(* IEC 61131-3 sources: ml2plc/benchmarks/st (part 23) *)

    bias_3 : ARRAY[0..63] OF REAL := [-0.00983189233, 0.0739286318, -0.03035645, 0.0550533831, -0.011248054, 0, -0.0295825377, -0.0090773385, 0, -0.0277472436, -0.00766381249, -0.00870534033, -0.0367787257, -0.0242641736, -0.00147182879, -0.00894620363, 0.0173237566, 0.00239057303, -0.00620334735, -0.00517789647, -0.0133990953, 0.0294917747, 0.0401097015, -0.0258607231, -0.00522571057, 0, -0.0150696058, 0.0860590115, -0.0117668696, 0.065539062, -0.00745888008, -0.0186666064, -0.010953215, -0.0240848884, -0.0448102988, -0.0404310934, 0.0785407722, 0.0790930837, -0.0278634299, -0.0265457965, 0, -0.0240220856, 0.00635804934, 0.0217319299, -0.02775204, 0.00820828322, 0.0399322994, 0.0746404901, -0.0329935588, 0, 0.00812079571, -0.0131024169, -0.0233938117, 0.0117759928, 0.0732261613, -0.0248215012, 0, 0.000535005063, 0.0062644016, 0.0363470353, 0.0787089318, -0.0285863206, 0, 0.0387545452];

    weights_6 : ARRAY[0..4095] OF REAL := [-0.0211104695, 0.157233626, 0.0721651465, -0.0791621804, -0.145463645, 0.0476885587, 0.103807047, -0.217098057, 0.15736191, -0.173330665, -0.128692865, -0.0421262085, 0.0980989784, 0.155999586, 0.0207046866, 0.184844807, -0.00715442142, 0.172988996, -0.206348658, 0.157887205, -0.037524119, -0.140499547, 0.187242225, 0.152909175, -0.145436138, -0.0675008371, 0.169665024, 0.210023656, 0.206236467, 0.208556831, 0.0959817022, -0.148986042, 0.0728623122, 0.026120171, 0.211910024, -0.0622561015, 0.0902522206, 0.0471122339, 0.0779013783, 0.0172086973, -0.039685376, -0.0467820168, 0.0570690036, 0.0242511332, -0.209991112, 0.00939850137, 0.112361535, 0.116925567, -0.153550565, 0.212469026, 0.14040117, -0.0208477583, 0.182546362, 0.0197014436, 0.186374202, -0.168809876, 0.196177915, -0.00232131779, 0.137093261, 0.162052512, 0.199661002, 0.0766961128, 0.211054429, 0.125300422, 0.00426613819, 0.288283914, -0.159290671, -0.0769464672, 0.0940423161, -0.0546351485, 0.0653043687, 0.0303289033, 0.0641354099, -0.192860484, 0.04200764, 0.0343205296, 0.155289501, -0.180832982, -0.12778616, 0.262020022, 0.0602597371, 0.10863255, -0.237889618, -0.095524922, -0.272757202, -0.0731869787, -0.0907882899, -0.147379801, -0.169592246, 0.178864881, -0.101507559, -0.0397703201, 0.016668126, 0.0635820627, 0.0767925531, -0.102012202, 0.0477126874, 0.0524956584, 0.111083403, -0.0878348276, 0.011967063, -0.0565153994, 0.170608982, 0.309960365, -0.105272628, 0.211850211, -0.0994742885, -0.153632715, 0.267046332, -0.203152657, -0.160044357, 0.0353948474, -0.0975862592, -0.0403899029, 0.07099244, 0.0249471422, -0.0422067828, -0.220276818, -0.185284197, -0.0370966718, 0.148172244, -0.120848358, -0.0141801946, -0.0953512639, -0.253198028, 0.104871087, 0.0740961581, -0.182465032, 0.0539166033, -0.159959942, -0.161966518, 0.0288212746, -0.135103494, -0.112145692, -0.0749802366, -0.0615305528, 0.157502532, 0.0857658535, -0.0273212269, 0.141590878, -0.0330497138, 0.176339731, -0.0418806784, 0.0999175385, -0.0713153332, 0.263013691, -0.115717605, 0.204661101, -0.11504811, -0.0947428197, 0.153199002, 0.335939616, -0.00631709397, 0.100122802, -0.209013268, 0.0137379616, -0.204656497, 0.0605559498, -0.175298169, -0.123451911, -0.0473049544, 0.0416926257, 0.156591177, -0.101554133, 0.115582488, -0.0190878287, -0.0975746512, 0.155756831, 0.108877532, 0.171931863, 0.235213891, 0.00560221262, -0.151249588, 0.00370491436, -0.0536345989, -0.181572989, -0.117012545, -0.106260225, 0.242837548, 0.223648071, 0.0628157556, 0.295081288, -0.0346996188, 0.15143846, 0.187727511, 0.290291816, 0.0033030943, -0.161266476, 0.00898908544, 0.244648784, -0.134097993, 0.0367004983, 0.0216495004, 0.180981815, -0.0798874199, 0.13122049, 0.0334438831, 0.0200074967, 0.103910699, -0.102675296, -0.207296401, 0.0869636759, -0.20655781, -0.0956464559, -0.203777537, -0.105265148, 0.0783180222, -0.0458374731, 0.204411358, 0.118474796, 0.122315288, -0.0419053994, -0.340604126, 0.135242134, -0.129586041, -0.0497838371, -0.0099619776, -0.0477824807, 0.281962305, 0.00426848233, -0.181631833, -0.170377254, 0.104996637, 0.114299156, -0.163810551, 0.249239355, -0.0833768472, 0.0697716847, 0.014485863, 0.157567188, 0.110193223, 0.230861947, -0.110680073, -0.0243154187, -0.0779362693, -0.0843363702, -0.049658794, -0.00124949845, -0.0668900907, 0.086151801, 0.179528475, 0.0938131064, -0.204934552, 0.0532739088, -0.120318048, -0.151893049, -0.146782264, 0.312886775, 0.0673337728, -0.1004811, -0.171645507, 0.268849701, -0.229744852, -0.134535402, -0.119718812, 0.0152729712, -0.196205392, -0.123321056, 0.00104016194, 0.114403293, -0.109209985, -0.116009399, -0.00587476185, -0.100333177, 0.104191698, 0.0102303922, -0.134384453, -0.204718813, 0.0862976313, 0.140776381, 0.0467067696, 0.094970122, -0.189605281, -0.0276639797, -0.0749640316, 0.0723377988, 0.00538966572, 0.0190833975, -0.0198820475, -0.00954220816, 0.0676214248, 0.104344197, -0.200903356, -0.206617773, 0.084322378, -0.0795044377, -0.0956577435, 0.191447124, -0.0795495212, -0.00805467833, 0.205130324, 0.179273605, -0.0990068316, -0.0614028908, 0.148120746, 0.132912666, -0.189888284, 0.200087667, -0.164052576, -0.0751432627, 0.0476862341, 0.0292347074, -0.052457124, -0.0892619789, 0.0716815516, 0.0529787801, 0.213911965, 0.209351331, -0.129100218, 0.0809682086, 0.176059052, 0.149538949, -0.126543701, -0.188590631, -0.183877945, 0.117343932, -0.167362183, -0.0124702444, -0.152586102, -0.18852441, 0.0780072361, -0.153538495, 0.0840239376, -0.148158073, 0.0951781124, -0.0676086247, -0.202492416, -0.0601291209, 0.0147494972, -0.148133397, -0.00998263061, -0.096799612, -0.00623972714, -0.0822741985, 0.134943768, 0.196010545, 0.0348980874, 0.194250599, 0.00896206498, -0.170046642, 0.0372118801, 0.0163984746, 0.179545149, 0.112079129, -0.104169428, -0.0681873262, -0.14190802, -0.167659834, 0.171136335, 0.176123098, 0.15911971, -0.0608612299, -0.0210849196, -0.132437974, 0.0952331275, -0.0566280484, -0.179609761, -0.202228233, 0.160658821, -0.127846152, -0.169803977, 0.0259776413, -0.175173402, 0.108989462, -0.174509123, 0.163906083, -0.0123733133, -0.192176595, 0.168579057, 0.167967841, -0.0916754827, -0.00778664649, -0.041722253, -0.215875, 0.107255802, 0.09431611, 0.110112235, 0.155124173, -0.0552193671, -0.00624886155, -0.116997302, 0.125487968, 0.149071887, 0.0814684778, -0.0264531672, -0.202291474, -0.107270196, 0.208046228, 0.198929116, 0.124986812, -0.116254002, 0.106430285, 0.0689994991, 0.123037621, -0.144080907, 0.0291826203, -0.0867067724, -0.122828558, -0.193552107, 0.180794746, -0.151306659, -0.108268835, 0.0360157453, -0.162983239, 0.180829659, 0.123341292, -0.143707618, -0.0218093451, 0.100755021, 0.048000399, 0.0416897722, -0.030838713, -0.10653317, 0.0873832777, -0.188493058, -0.0422797352, 0.0743354112, -0.125618383, 0.163786501, -0.184897706, 0.0689249486, 0.216842949, -0.173285306, 0.185100108, -0.117793359, -0.19082053, -0.106456965, -0.0742470324, -0.0494265445, 0.165998891, -0.185700104, -0.121370681, -0.174497947, -0.0514864251, 0.10049998, -0.107571743, 0.159631327, 0.187085122, 0.0653448254, -0.120375261, 0.275558501, 0.182469591, -0.175698802, -0.0759939849, 0.065009132, 0.259765774, -0.086910978, 0.0502287, -0.0737552643, -0.0215020366, 0.161072969, 0.123396195, -0.175406262, 0.0518808141, -0.0351930261, 0.0470791981, 0.262363374, 0.1363094, 0.180866018, 0.132682219, 0.165143073, 0.126118854, 0.0938046128, -0.254130632, 0.0568571538, -0.0724096671, 0.0160691887, -0.0521572456, 0.22484374, -0.0792442709, -0.00761091337, 0.276181072, -0.086371094, -0.129833862, -0.0362726077, -0.0417017639, 0.0206526667, 0.239292666, -0.0601968914, 0.0359402746, 0.308184862, 0.0270620137, -0.208643079, 0.131217003, 0.0645703152, 0.118619733, 0.0201364737, -0.165239125, 0.162001967, 0.177479923, -0.111770749, 0.135645315, 0.0129162921, -0.202752113, -0.0295399278, 0.022838518, -0.0796107128, 0.0467211269, -0.051113341, 0.160861671, 0.00665348954, -0.104955673, -0.0838543624, -0.236661151, 0.214804575, -0.0623946115, 0.140443742, -0.0886547342, 0.0746734887, 0.276039749, -0.199886113, 0.121124074, 0.0216602683, -0.167079479, -0.138646215, -0.0189068019, -0.0126770437, 0.0390007943, 0.0360741764, -0.141568631, -0.0118533075, 0.178898349, -0.0807059556, 0.0550475866, 0.178213313, -0.0915158764, -0.109646633, -0.066618517, -0.00931756198, -0.201538652, 0.0959077924, -0.019727543, 0.00191234052, 0.180038348, 0.112552777, 0.101054952, 0.215217724, -0.185405463, 0.122277573, -0.0108845085, -0.0374378562, -0.0693836063, 0.206913039, -0.193783402, -0.0592647493, -0.198673338, -0.00192482769, -0.00480589271, 0.0151784569, -0.11449635, 0.150387093, -0.0220891237, -0.0531173348, 0.0558237582, -0.0155561566, 0.110152856, -0.10219758, 0.125887617, 0.187418178, -0.00413711369, 0.199766979, -0.0751423836, -0.196204484, -0.163247168, 0.0657932907, 0.179478303, -0.0909180194, -0.0187031627, -0.0687615424, -0.125233293, -0.00715054572, 0.191343263, -0.140845746, -0.101612061, 0.028948009, 0.00607836246, 0.0241835825, -0.0792405158, 0.170693278, 0.121472552, -0.159257323, 0.15754503, -0.139394745, -0.044453688, -0.0742065012, 0.176449284, 0.226904213, -0.0162550025, 0.281962007, 0.141561612, -0.179304242, -0.22687985, 0.0888308734, 0.1368251, -0.215948135, 0.232278898, 0.14440532, -0.210397243, 0.0025057646, 0.257558495, 0.069859311, -0.0588960908, -0.178999975, -0.00917844474, 0.0827753693, -0.0334500261, 0.0289534777, -0.147056982, 0.18982479, -0.0401569977, -0.00673311763, 0.117641859, 0.0199112538, -0.110949092, -0.10525246, -0.110742055, -0.149034083, 0.176191643, 0.164675817, -0.152210981, 0.111859016, -0.0424617529, 0.070398286, 0.0940225571, 0.160483241, -0.166004077, -0.0361319557, 0.156162739, 0.255399585, -0.0411905348, 0.0899951607, -0.214364231, -0.0514262058, 0.136874646, -0.0144281425, 0.0158658996, 0.173274562, -0.0837578475, -0.021164313, 0.189715445, 0.0227939058, 0.0768007636, 0.0420344919, 0.13114506, 0.0212835968, 0.125271335, -0.0908199325, -0.2127489, 0.223346874, -0.168397516, -0.143092021, 0.0855721906, 0.217426375, -0.010913834, 0.161978483, -0.0237388425, -0.0148029672, -0.0206773132, 0.163911536, -0.115519904, -0.0708635896, 0.160120934, 0.21680361, -0.0919932425, -0.106572457, 0.186694637, -0.0864723846, -0.0672358871, -0.0620637983, -0.0492999963, -0.031213671, -0.214064613, -0.0040052929, -0.177249506, 0.198898122, 0.029973764, 0.0648880824, -0.0722419471, 0.0583239459, -0.161417127, 0.118529066, 0.0775398463, 0.0136581725, -0.019831283, 0.0340036228, -0.069475472, -0.141518444, -0.0155703966, 0.0465259701, -0.13712129, 0.215217024, 0.153940856, 0.233599231, 0.069659397, 0.0283375084, 0.136588395, 0.114837028, 0.00435284665, -0.0815577209, 0.0850224197, 0.0896461308, 0.0839098245, 0.12630628, 0.102898523, -0.0242574364, 0.0395214707, 0.179158911, 0.140869483, -0.0315961689, -0.211324051, -0.101073779, 0.164895773, 0.0432892777, -0.0961784273, 0.187965691, -0.0886578932, -0.143109977, -0.200058162, 0.128884479, -0.150142565, -0.0212808698, -0.0118450765, 0.0831215233, -0.0732853338, -0.0489297211, 0.000687902851, 0.0266030431, -0.201587737, -0.185360029, -0.00679598097, 0.108024552, 0.102891639, -0.178852096, -0.173995063, 0.0813450366, -0.0506051332, -0.0515105948, 0.0880956501, 0.173789188, 0.00271931873, -0.181898132, -0.0750331804, -0.0916771367, 0.0279746372, -0.0858160108, 0.0492289215, -0.0897664428, 0.118924871, -0.00673155487, 0.0254511833, -0.0507416576, -0.131477594, 0.0658444315, -0.176156193, 0.00369836204, 0.209861919, -0.144315973, 0.0758810192, -0.126617879, 0.0478404015, 0.0629696399, -0.181336939, -0.070628196, 0.0589700602, 0.0671523064, 0.0530530922, 0.148497984, 0.199353352, -0.2551274, -0.155184016, -0.00421486888, 0.212831467, -0.0586378425, 0.147449061, -0.201066777, -0.0765811056, 0.0298376996, -0.028335914, -0.0145538365, 0.120011285, 0.263296843, -0.0805929601, 0.196454912, -0.194894016, 0.0144730853, 0.00976360589, 0.105623856, -0.128629684, 0.224141806, -0.244979411, 0.214529052, -0.0382702313, 0.156628206, 0.0189788435, 0.127576098, -0.204321966, -0.106341101, 0.309783638, -0.0312428474, -0.136540458, 0.271282047, -0.320485145, -0.130114317, 0.0987244472, -0.0768140033, 0.292481333, 0.028581921, 0.0651605949, 0.0565245636, -0.207960293, -0.105757877, -0.0665429085, -0.00274416106, 0.0682443231, -0.106524602, -0.163970143, 0.0532483347, -0.200977892, 0.0309002809, -0.0602365695, 0.202884033, -0.04036038, -0.0263917297, -0.138741806, 0.261350095, 0.0551347472, 0.181741431, -0.147500739, 0.178088039, 0.114219822, 0.046044156, 0.0941443816, 0.0813267976, 0.0595558062, -0.197245672, -0.0100678066, -0.211604849, -0.148000121, -0.198542699, 0.196343526, 0.138460979, 0.107107386, 0.0907673761, -0.121037595, 0.252360672, -0.0970465541, 0.0558764599, -0.0847656652, -0.209763199, 0.167329192, -0.237716049, -0.0499278046, 0.249167144, 0.0408127345, -0.165352255, 0.176838875, 0.00782003999, 0.176427022, -0.0851962119, -0.192636058, 0.187963501, 0.170646742, 0.0470952839, 0.00458228588, 0.141556203, 0.0644658133, 0.0417393818, 0.0441780165, 0.039651297, 0.0833919719, -0.172924563, 0.0634429529, -0.0965564921, 0.0724875107, 0.21937269, -0.0974312797, -0.130002752, -0.121189877, 0.0671949536, 0.0867445171, -0.00312029221, 0.126738116, 0.0653212741, 0.252740234, 0.287628323, 0.167519346, 0.139367387, -0.0309090856, 0.263746917, 0.0875785947, 0.0128881168, -0.0565036125, 0.120908678, 0.240472659, -0.201509178, 0.293792278, -0.131671205, 0.0896654353, 0.0370695144, 0.135521129, 0.20480074, -0.175205469, -0.171041086, -0.0579688512, -0.156582564, -0.0778886229, 0.0664458051, 0.130356193, 0.0996769667, -0.153313071, -0.192398816, -0.106274486, -0.0162558295, 0.0870158821, -0.192340657, 0.048169598, -0.171457037, -0.136983603, -0.064907901, 0.145346314, 0.190712199, 0.0360278338, 0.0434320495, -0.211738184, 0.160129383, -0.105414405, -0.171388596, -0.0388856754, 0.142384306, 0.137329713, -0.130360201, -0.0619715676, 0.00965698808, -0.0439127162, 0.170497492, 0.212079838, -0.142104536, 0.0586519986, -0.115233481, -0.0224351734, -0.16999881, 0.0918107182, -0.167155147, 0.195335492, -0.0757286102, -0.172540411, 0.103915311, -0.141615734, -0.00377908791, -0.0657154992, -0.148804039, 0.022908235, -0.168834493, 0.152186722, 0.0506493412, -0.112933271, 0.00049599976, 0.100557655, 0.112081513, 0.142245606, 0.0271094441, 0.0381551534, 0.20742555, -0.110420324, -0.100627325, 0.145201087, -0.202350944, 0.120480955, 0.0444104783, 0.211891606, 0.19280535, 0.0655445755, 0.189393878, 0.196804807, -0.0521670766, 0.0503715128, 0.214662924, -0.0492795333, -0.0675857663, 0.178876325, 0.0826835707, -0.169171751, 0.0269653201, 0.211806223, 0.130338058, -0.000949479057, 0.196632594, 0.186210766, 0.0524837524, -0.0555000752, -0.131404147, 0.146059439, -0.0972863659, -0.0147773847, 0.105667993, -0.00656548562, -0.144193918, 0.0886233747, 0.215485469, -0.0223604683, 0.165627271, 0.117518991, 0.000273500162, -0.196279138, 0.0528765172, 0.137227044, 0.0115529299, -0.0449971259, -0.0784725025, -0.172097519, -0.0769113824, -0.144809157, 0.087641567, 0.0567293391, -0.165308416, 0.0845244378, -0.0673978627, 0.191283584, -0.0394614935, 0.203768536, -0.202162296, -0.138682559, -0.109796427, 0.112647042, 0.0804700181, -0.0721322224, -0.102790877, -0.0195402578, 0.00424019992, -0.117378324, 0.205446005, 0.203034252, 0.101452544, -0.0454550199, 0.157199964, 0.0115054222, -0.0943236724, -0.0565667748, -0.107933104, -0.0655731708, 0.157481402, 0.128197148, 0.00223283307, -0.00375899929, -0.1018316, -0.173439905, -0.15236567, 0.212863877, -0.152796358, 0.162461266, -0.0564482771, -0.120488144, -0.13375029, 0.025584979, -0.205807254, -0.192222401, 0.214670464, -0.0954632461, 0.183467418, 0.183182776, -0.00882993639, 0.169890597, -0.197005555, -0.106948674, -0.00395756867, 0.0120129455, 0.0223759171, 0.149836347, 0.228335664, -0.0534032434, 0.132094547, -0.0133346152, 0.183536708, -0.190487862, -0.00259809522, 0.000128543412, 0.127965212, -0.0134203611, -0.129633933, 0.229406625, 0.0699569285, 0.198570237, -0.0478203781, 0.181146488, 0.0680752471, 0.00578152016, -0.110974222, -0.088077426, 0.117438272, -0.202719942, -0.0765619129, 0.0070055034, 0.00518807769, 0.0908474326, -0.210115537, -0.259739071, 0.0877127647, 0.178909853, 0.0252563711, 0.161810607, 0.14697203, 0.0207887739, 0.192217827, 0.0119345486, 0.111504808, -0.138566241, 0.0183499251, 0.178135261, 0.10215006, 0.11800538, 0.0883670896, 0.0227976646, -0.122666731, 0.0188208688, 0.0996467769, -0.100148812, 0.117532745, 0.237992808, -0.130577683, -0.15731205, 0.271030456, -0.23369348, -0.0929943994, 0.0971348509, -0.104811274, -0.120445482, -0.0412788987, 0.0163263902, 0.138564199, -0.144116297, 0.125310749, -0.172860175, -0.224062487, 0.13113521, -0.0350915194, 0.102414116, 0.00754255336, -0.0123361535, -0.0915403515, 0.0783033222, 0.109218769, 0.00511339353, 0.059927389, 0.0361303464, -0.121367157, -0.0622647256, 0.0529602021, -0.149987593, 0.0344639942, 0.244372755, -0.129179358, -0.0458081402, -0.141225874, -0.00293263793, 0.152275071, -0.0406294242, 0.139919147, 0.187548757, -0.178822875, -0.0349252298, -0.0637998432, -0.192398965, 0.0176388826, 0.0132232755, 0.081162639, 0.00220011175, -0.148068249, 0.189775273, -0.21044074, -0.193314359, -0.0609930158, -0.191583186, 0.169178709, 0.170702919, 0.149429336, 0.0734934062, -0.0319855362, 0.0536946096, 0.0498708934, -0.117750682, 0.0036894232, 0.0974819437, 0.162416473, 0.036212638, -0.152097091, 0.0102473954, -0.175146922, -0.109410793, 0.0510285608, -0.102032453, -0.0270780027, 0.112112477, 0.179075554, -0.174917683, -0.115047842, -0.104785867, 0.0759669393, -0.185626954, -0.114752382, 0.0533825904, -0.104991615, -0.0954450741, -0.0869510844, -0.132044673, -0.191752613, 0.00513811922, 0.0554652661, -0.133202344, 0.148236826, -0.174548671, 0.101005033, -0.147775263, 0.151600003, 0.195948124, 0.146968648, -0.181632847, -0.126265585, 0.0861280486, 0.0299651623, 0.0794558972, 0.0533921868, 0.0195937455, 0.0455982238, 0.150372431, 0.139378235, -0.101709567, -0.0294380337, 0.0811925083, -0.0342354178, 0.0327691734, 0.0400085896, -0.1412265, 0.0617004111, 0.0421027988, -0.104852192, 0.00592757761, -0.180350497, 0.0525539964, -0.111471675, -0.0811403841, -0.0120081007, 0.15921399, -0.188091248, 0.184693262, -0.0228968561, 0.115342319, -0.0535733849, -0.114198565, 0.0240756273, 0.147423342, 0.15892826, 0.00908050407, -0.213146105, 0.152774766, -0.00141887786, -0.0586975515, -0.114548035, 0.0891831964, -0.0406573191, 0.0181619823, -0.049714718, -0.200603843, -0.135449693, 0.129440948, -0.212808505, -0.0500480942, -0.0812454671, -0.180212289, 0.0619920045, 0.0307168979, -0.0518378466, 0.0701079816, -0.190243214, -0.138796121, -0.193981051, -0.0390182026, -0.117929213, -0.204903558, -0.202367961, -0.155948266, -0.171265543, -0.129201606, -0.0976203829, 0.221453071, 0.138735101, -0.158441961, -0.225554422, -0.0675398037, -0.132319763, -0.0978091806, 0.210110873, 0.178208128, 0.101490974, 0.0418321043, 0.160106704, -0.187610939, -0.192003295, 0.0196090881, 0.0968832597, -0.175496653, -0.0902556181, -0.155951157, 0.107045144, 0.0573832281, -0.0581211299, 0.0521087125, 0.171671689, 0.158271715, -0.212730348, -0.0388053134, -0.172507182, -0.125131086, 0.156479985, -0.335062623, -0.0702413097, 0.223254368, 0.0645823479, 0.219279632, -0.196573928, 0.0732722208, 0.263311893, -0.159265086, 0.0834448114, 0.13835384, -0.136304572, 0.106453225, -0.0613590926, 0.138230368, 0.174712658, 0.094565548, 0.0211733319, 0.102425985, 0.0467876047, 0.111685343, 0.147267804, -0.258844495, 0.145146266, 0.14244695, -0.22259891, 0.0884163454, -0.207033977, 0.202475429, 0.0740721077, -0.0818101689, -0.125599563, 0.048894804, 0.139541343, 0.0525139496, -0.179559693, -0.0716978014, 0.0090209581, 0.113008924, 0.172887772, -0.0844542906, -0.0717213899, 0.188895106, 0.00843533594, -0.161318779, -0.00458678044, 0.0416456424, 0.0458753034, -0.117116317, 0.134884998, -0.0610275529, -0.0735569224, 0.220500335, -0.0618452467, 0.0568264462, 0.0672242194, 0.0536397211, -0.0376431644, 0.156504616, -0.207624599, -0.0204942245, -0.208658844, -0.179129675, -0.100364596, -0.150991708, -0.186092764, 0.17417559, 0.134831354, -0.095172435, -0.0442455336, 0.256724715, 0.21277459, 0.17345655, 0.216043293, -0.0360164866, -0.0652590916, 0.0154270008, -0.0202574134, -0.175363034, 0.0316524692, -0.0490601547, -0.0729391202, 0.13120921, -0.115910649, 0.162211448, -0.200046033, 0.113587596, -0.098146148, -0.062560007, -0.212389871, 0.212651432, -0.207820579, 0.16756323, -0.120097443, 0.245886236, 0.0261694063, 0.250802189, 0.213231578, -0.110681944, -0.0259542018, 0.0393911712, 0.141605258, 0.0951679051, -0.0903783441, 0.0266120266, 0.130146444, -0.202337459, 0.0765965804, -0.010533765, -0.0858198181, -0.00901217386, -0.0870363861, -0.011424928, -0.090558961, 0.0835403949, -0.256125689, 0.0130133061, -0.127759323, -0.238343403, 0.161234543, -0.192689836, 0.27777794, -0.0743051767, -0.0246492773, -0.264801741, 0.13777788, 0.039771352, -0.199020803, 0.278468162, -0.208027422, -0.0828270987, -0.00967502873, -0.0816069394, -0.0424416326, 0.0527059995, -0.163091287, 0.00891038775, -0.224737093, -0.0790355057, 0.0459024347, -0.0678463578, 0.174242303, 0.00127267418, -0.0481367819, -0.149950892, -0.261374563, 0.152924955, 0.115787119, -0.151344597, -0.208144918, 0.193755448, 0.148202732, -0.200177088, -0.14347811, 0.0296298023, 0.120643049, 0.0740528107, 0.0289400071, -0.219525307, -0.0684371665, 0.170777753, 0.0165751912, 0.161401957, 0.09001939, 0.137214094, -0.0132981138, -0.075612478, 0.223878801, -0.129973829, 0.163486749, 0.025689736, -0.02602401, -0.176745981, -0.096706301, -0.229914978, -0.208292037, 0.115179032, 0.131318823, 0.12323276, 0.0363375023, -0.18000105, 0.0444394164, 0.292281061, -0.209439784, -0.0804421529, -0.241354913, 0.0492477566, 0.115014032, 0.113993555, 0.0711855739, -0.105379127, 0.116060019, -0.230782375, -0.071728304, 0.166753724, 0.141988203, 0.203238681, 0.135525316, -0.0675361156, 0.258204639, 0.0555558056, -0.0669079423, -0.0546362698, -0.0095171025, -0.112937562, -0.112366028, 0.196951315, -0.190239713, 0.100786179, 0.27030012, 0.0785356015, 0.0146926921, 0.0336835608, -0.0475944877, -0.25933221, 0.114190906, 0.159268126, -0.0437385812, -0.259978563, 0.119038261, 0.196310908, 0.126920417, 0.1142755, 0.0501057506, 0.134804621, -0.0957523063, 0.14846307, -0.0672448725, -0.16493322, -0.21647732, -0.138321653, -0.0105587812, -0.105590709, -0.183317751, -0.0017683208, 0.0214145966, 0.0840778798, 0.1456929, -0.141866982, -0.177974984, -0.183813006, 0.0323574543, 0.216028988, -0.174554035, 0.0929575935, -0.0752552748, 0.0173932761, 0.00922764838, -0.194893017, 0.129454538, 0.132133171, 0.13402985, -0.0701206028, 0.176784858, -0.0571110547, -0.0514186881, -0.08907713, -0.0646748692, -0.194243208, 0.129443407, 0.00619410118, -0.00450532138, -0.207810163, 0.0717498884, -0.0734594464, 0.124055974, 0.075352475, -0.150470659, -0.187533662, -0.0271674097, 0.153355226, -0.0271843374, 0.0681567341, -0.0659090728, -0.0516456589, -0.198433399, -0.0102793267, 0.0921462923, -0.107441001, -0.0820229352, 0.0697086006, -0.121913351, -0.0349813551, -0.0305808745, -0.0559222177, -0.0764169097, 0.170531899, -0.119125612, 0.0380934328, -0.0192875862, 0.0188238919, -0.0392661095, -0.202440292, -0.115953766, -0.132373601, 0.210289285, -0.207067996, -0.074820444, 0.171109334, -0.0611716658, -0.187234789, -0.178964883, -0.0744869262, 0.042780444, 0.0340865999, 0.0349340886, -0.0808666945, 0.200756922, -0.0821405053, -0.177407742, -0.0506182462, 0.0319291204, 0.111412361, -0.119748138, 0.0575083643, 0.148518518, -0.0711778849, 0.0900242478, -0.166702032, 0.0707694143, -0.0672384202, -0.148692697, 0.0733167678, -0.0461998433, 0.0212943405, -0.105709076, 0.0511011332, -0.0303771347, 0.0363206118, 0.0554131418, -0.191839933, 0.0704303831, -0.014075771, -0.192795038, 0.0864057988, 0.0957165509, 0.0517887622, -0.207105055, -0.0549096018, -0.197128266, -0.0435425937, -0.00281360745, -0.0405648947, 0.0581579953, 0.131218538, -0.16994527, 0.199992672, 0.115575358, -0.18995063, -0.156800047, -0.0196557939, 0.076645188, -0.163925126, -0.123550206, -0.00278422958, 0.0024073571, -0.075328432, 0.0587575585, 0.194733024, -0.112012841, -0.17458263, 0.0873643756, -0.171549991, -0.150170997, 0.145191774, 0.0886108205, -0.191762626, -0.102553405, -0.103013307, -0.116796724, 0.200971395, -0.162655994, 0.0177573599, 0.0770139471, 0.135249302, -0.149339631, 0.0532134771, 0.125556737, -0.111500844, 0.13430278, 0.116502553, -0.133535191, 0.0993374139, 0.0131562548, 0.141030326, -0.215099677, -0.0540164895, 0.0587758832, 0.133371785, 0.128054485, 0.181748942, 0.186617449, 0.140814275, 0.158420652, 0.117290303, -0.0828610957, 0.181842074, 0.0536724478, -0.156423688, -0.0572760254, -0.0758121386, 0.0171979927, 0.0617454574, -0.123269998, -0.0501214638, 0.210173443, -0.0469620526, -0.0736155212, -0.0198381282, 0.159689367, -0.164338425, -0.148481369, -0.0429480225, -0.0946798697, 0.200503424, -0.101595551, 0.201301143, -0.0489229187, -0.162824064, -0.0438856035, -0.21362631, 0.244266868, 0.274435222, 0.169392526, -0.185727969, -0.0522047542, 0.00556242652, 0.0991317555, -0.132557571, 0.172653839, 0.0851856023, 0.190462366, -0.117255479, 0.117573619, -0.132007942, -0.0157813504, -0.00529545965, 0.0486687161, 0.209120095, 0.188496932, -0.197368637, 0.0993192643, -0.154122457, -0.135731071, 0.0958589017, -0.109322362, 0.0503121465, 0.0242886506, -0.151156679, -0.141134143, 0.0115236547, -0.248438224, -0.112202108, -0.0897251442, 0.253748894, -0.000320830557, -0.138551369, -0.0638582781, -0.0156727377, -0.10645014, -0.000941439182, -0.117576726, 0.0970672369, 0.159923315, 0.136554152, -0.0385889336, -0.103830874, 0.0358882025, -0.187269032, -0.206554636, 0.0885479078, -0.0132518057, 0.214956224, -0.12615642, 0.275876939, -0.0640837476, 0.144479454, 0.205591425, -0.0275788121, -0.140130028, 0.203447714, -0.107345656, 0.177566424, -0.112334542, 0.135879055, -0.141970098, 0.109072447, 0.110946029, 0.10664539, -0.176637948, -0.212433696, 0.0630291849, 0.150753275, -0.124068864, 0.0347972997, -0.203520656, -0.162690356, 0.0804221854, -0.183624178, -0.168030873, -0.0466670021, 0.201229915, 0.0762459859, 0.0738973469, -0.107046053, -0.0266148597, 0.140076771, 0.0768975466, -0.0661414787, 0.205275372, 0.117615834, 0.162698045, 0.0471834056, 0.066787824, 0.0462587886, -0.0657628477, 0.150616497, 0.180957869, 0.0334356651, 0.0815333351, 0.182552829, 0.0747729093, -0.0848053396, -0.192697644, 0.000992957503, 0.0669444054, -0.0864309072, -0.208967999, -0.163346067, 0.0919444114, -0.11361666, 0.0901513845, 0.121801101, 0.18307288, -0.129042506, -0.0295936447, 0.133450344, -0.149377078, 0.0841869488, -0.167957082, -0.156804591, 0.111636445, 0.122521162, 0.0814686567, 0.0948956907, -0.142786413, -0.16495119, -0.0619355738, -0.151000232, 0.235567585, 0.242622092, 0.0626911446, 0.158189178, -0.130945265, -0.0510335267, -0.193246707, 0.181436405, 0.039453797, 0.0719453469, 0.000969689456, -0.204767287, -0.0541508645, -0.0104957288, -0.165310189, 0.228289202, -0.133238673, -0.173104972, -0.197261706, -0.160179675, 0.207100019, -0.20425573, 0.0656981021, -0.064999491, -0.0689243972, -0.0135737462, -0.114986956, -0.148001194, -0.156635731, 0.136174291, -0.0735397115, 0.024009943, 0.18861106, -0.0555349216, 0.167080164, -0.0663658902, 0.156313211, -0.137416631, 0.219937623, -0.0101457722, -0.192980722, -0.00603267178, -0.00608571619, 0.156647861, -0.213914216, -0.00686631678, -0.18698661, 0.137742862, 0.107735321, 0.0747293308, 0.135365367, -0.0309074614, -0.103391051, 0.253569245, -0.167082265, -0.155858532, -0.0525114238, -0.182957605, 0.192761794, -0.103556834, -0.0391536839, -0.0144170625, 0.179714397, 0.0125448611, 0.164514452, 0.108714201, 0.228309497, -0.086764805, -0.134017855, -0.0286707878, 0.0568587519, 0.081173256, -0.0287004691, -0.0670309067, -0.064888604, 0.114137292, -0.0725059435, -0.174008653, -0.0875643715, -0.127273753, 0.131509304, 0.225763783, -0.0839330703, -0.136040702, -0.189437702, -0.202584773, 0.0523217767, 0.263796657, 0.136124715, -0.175133616, 0.0481774323, 0.0252242032, 0.180632174, 0.14017573, 0.0722272471, -0.141429991, -0.14743869, 0.172693461, 0.250584245, -0.0508589484, 0.149392784, -0.0614273623, -0.188037321, 0.136032209, -0.115289845, -0.215180367, 0.175799161, -0.142253354, 0.0276352465, -0.149539113, -0.0436008498, 0.214859545, 0.134571746, -0.0436521098, 0.222684115, -0.109537765, -0.0431752317, -0.0141235311, -0.0353392698, 0.182102561, -0.152115494, 0.237127289, -0.166017041, -0.0662677586, -0.123375967, 0.0391481966, -0.0662866086, -0.032407172, -0.226494104, -0.163152546, 0.00762933912, -0.171422973, 0.25206548, -0.0176769458, 0.277596235, 0.00642719865, -0.0545174591, 0.0522982441, -0.0763136446, 0.245492265, -0.0421209559, -0.140477717, 0.123090878, -0.069406189, -0.00897048693, 0.0338697173, -0.145748019, -0.143358067, -0.170915663, 0.179273531, 0.0158482641, 0.0439317264, -0.164723992, -0.163618878, 0.129824698, -0.307914853, 0.00500768237, -0.177501172, -0.196434334, 0.159178451, 0.193265259, -0.0784411952, -0.0199198276, -0.136541232, -0.0581868403, -0.0336628743, -0.163134873, 0.0191420875, 0.00514668226, -0.136096939, 0.169880554, 0.146405965, 0.12389233, -0.157588914, 0.135902241, 0.020170236, -0.197500393, -0.211237401, 0.183388785, 0.173877329, 0.0596420616, -0.0495417826, -0.00247370661, 0.196426719, 0.119838014, 0.030950062, 0.0507870428, -0.0551843941, 0.080456607, 0.13434732, -0.188290507, -0.0291505717, 0.0936101824, -0.0743033737, 0.238530099, 0.0853732973, 0.0866866857, -0.0472731218, 0.101936914, -0.161955655, -0.103445411, -0.115826197, -0.185676217, 0.144468918, 0.0192127451, 0.243185744, 0.213160887, -0.0700132027, 0.132710531, -0.0866566449, -0.126810819, 0.239814758, -0.0543582328, -0.0970630199, 0.151953116, 0.247111589, -0.157347828, 0.137009367, 0.0681802928, -0.325023025, 0.0898184255, 0.0172431283, -0.0638230145, -0.00389597355, 0.201046601, -0.10115499, 0.215875402, 0.148981452, 0.156407848, 0.0929401219, -0.116457552, -0.0533874482, -0.0953917503, 0.0635540038, -0.174071953, -0.014446131, 0.174123392, -0.0109589575, -0.06459672, -0.00470030122, -0.210424423, -0.214112669, 0.073211208, -0.116393417, -0.215505868, 0.165930703, -0.111611903, 0.0542642213, 0.02777946, 0.254414827, -0.237083703, -0.106226139, 0.135093778, 0.188917518, -0.088959381, -0.153844506, -0.0671698377, -0.253456146, 0.211136952, -0.0188651383, 0.00893640518, -0.0500897728, -0.103367783, -0.209297687, 0.185887992, -0.0478939153, -0.121324107, 0.19026418, -0.0403532162, 0.206234485, 0.206992447, -0.200000763, 0.156136796, 0.0766848624, -0.213080689, 0.129118517, -0.0300498139, 0.0841510743, -0.0039588213, -0.053927239, 0.0600163192, 0.118532047, 0.125032127, -0.141252995, -0.134606391, -0.149302527, 0.181654245, -0.0525682978, -0.0095063895, -0.0866127312, 0.0237378366, -0.0967183784, 0.133381084, -0.0180076975, 0.0250853039, -0.159199923, 0.179142401, 0.146943107, -0.0130850719, -0.208270669, -0.122804597, 0.086103417, -0.0587755069, 0.140682414, -0.192945361, 0.0519251116, 0.232186466, 0.0842411444, 0.0156072173, -0.0367138796, -0.129091635, 0.286088198, -0.050661698, -0.0959331617, 0.196171507, -0.166134045, 0.110787347, 0.0763130635, -0.195894212, -0.016266359, 0.0650015101, -0.000705195009, -0.0798940808, -0.157687202, 0.0367488489, 0.0635683686, -0.00835195277, 0.147954598, 0.00347357406, -0.0717437714, 0.0263384692, -0.0868112966, -0.1464587, 0.183965608, 0.154775858, 0.0563162044, 0.119879685, -0.0458873212, 0.0146314949, 0.01340455, -0.127139658, -0.0805401057, 0.010805428, -0.0598547757, 0.140515849, -0.0332521386, -0.139405355, -0.00381903304, -0.119757995, 0.0642717928, -0.00595461437, 0.00971299782, 0.0181997381, 0.14657104, 0.236595348, 0.133447409, 0.165538937, -0.171264574, -0.17734462, -0.118777111, -0.0742687881, 0.163928539, 0.158281639, -0.0200940482, 0.00364433066, 0.110924534, 0.204607725, -0.056781482, 0.00452534854, 0.161825106, 0.231086031, -0.114858396, -0.00962379854, 0.207619533, 0.090628311, -0.0552490801, -0.168093532, 0.12639004, -0.0469605736, -0.124545485, 0.103754275, 0.116334625, -0.200652197, 0.122327343, -0.24620837, 0.150227144, 0.124391578, -0.149749219, 0.0835158229, -0.15222469, -0.0924759209, 0.121347412, 0.103715703, -0.179746136, 0.0542897433, -0.121789955, -0.0700749233, 0.0558092073, 0.159794122, 0.125659496, -0.0444125459, 0.0128017385, -0.172242373, 0.17140238, 0.0414437614, 0.0733803064, 0.0441474169, 0.0272179805, 0.0157027543, 0.0845738202, 0.19979848, -0.103852771, 0.145444691, 0.1565492, -0.183115691, 0.0272264779, 0.00203362154, -0.176931471, -0.136718005, -0.0667834654, 0.160385624, -0.0971334875, -0.0346084386, -0.00125173316, 0.214042053, 0.100500204, -0.181512147, -0.207882851, 0.18568328, 0.205129042, -0.012027801, 0.136106357, 0.0456399471, 0.181273654, 0.0196859818, 0.0653820038, 0.0663783401, -0.0337033458, -0.0586933829, 0.108097129, 0.091456309, -0.134444326, -0.027708875, -0.145242408, -0.00287574693, 0.0847207606, -0.181775391, 0.183636069, 0.0688786507, 0.263257593, -0.00427195895, 0.123155445, 0.158885136, 0.170019612, -0.181566104, -0.0179279, -0.184301853, -0.0013938545, 0.177570879, -0.121418886, 0.0150488978, -0.000610802672, -0.218872413, 0.133591279, 0.112349041, 0.202252939, -0.194210395, -0.0492385663, 0.199029937, -0.0331471264, -0.189999968, 0.15875043, -0.0649037361, -0.0359622762, -0.101073802, 0.178152233, 0.0650028139, 0.0732081607, -0.0311551392, -0.00686773099, -0.112522438, 0.281459391, -0.150038421, -0.154241458, 0.0597723648, -0.0180041976, 0.095261544, 0.196119681, -0.0852496773, -0.220084459, -0.141354889, -0.00177710166, 0.115805745, 0.211524799, -0.146760225, 0.130397364, -0.200928628, -0.082532011, -0.0342374705, 0.0937826261, 0.204201654, 0.259379774, 0.143860042, -0.022885045, -0.0885771513, 0.225629315, 0.203129902, -0.0972949266, -0.167454958, 0.209564671, -0.0261494219, -0.121619433, 0.170461625, -0.0545143932, 0.0480193757, 0.184107944, -0.127340436, 0.183212698, 0.121917456, 0.189465776, -0.198853567, 0.176508516, 0.0776296109, 0.071349591, -0.163570002, 0.121416613, 0.0280675068, -0.0353203863, 0.0381100923, -0.0884888694, -0.00105153024, 0.197435677, -0.0372472778, 0.199374154, -0.0266889483, 0.0552413613, 0.16077064, 0.0775329843, -0.056018278, -0.0785094425, -0.111316718, -0.0708481371, -0.219346598, -0.0713492781, 0.0917782038, -0.111492112, 0.0235726535, 0.113839343, -0.0846240744, 0.186591521, 0.107423566, -0.0425455049, 0.133113995, 0.112909913, 0.155081719, 0.12983717, -0.0908117145, -0.0424004309, 0.123853929, 0.161590233, 0.0740211159, 0.220889717, 0.0111323493, 0.0138287498, -0.108956374, 0.218805134, 0.116877005, 0.0139654735, 0.0478446335, 0.00290354271, -0.135019958, 0.100197278, 0.202663228, -0.0565481894, 0.0516312271, 0.164359331, 0.027229758, -0.161545083, -0.0841104686, -0.132132292, 0.0750347823, 0.126185328, -0.0328487605, 0.121280387, 0.17534402, 0.142205924, -0.222641334, -0.0284508038, 0.0550886728, 0.0873866901, -0.098779656, 0.108810529, 0.222481266, -0.133257478, -0.0171785951, 0.23207663, -0.16922313, 0.0166405141, 0.149411425, 0.244119301, -0.0342978686, 0.0424096137, 0.0300826505, -0.302469999, 0.12808831, 0.202303231, -0.128145292, 0.254153311, -0.0533468723, -0.00429165037, 0.00639062561, -0.0596186407, 0.106781147, 0.116036557, 0.164889902, 0.118450627, -0.11772456, -0.212542042, -0.0230301227, 0.15320763, -0.102894507, 0.164426908, 0.137734249, 0.0360440724, 0.053503558, -0.19689019, -0.089921236, 0.255165786, -0.121091068, -0.186938509, -0.199636534, 0.228079587, 0.0136816055, 0.137275338, 0.147264242, -0.157951266, -0.133595556, 0.198956296, 0.0500613302, -0.104482673, 0.153554499, 0.186254889, 0.0757497177, -0.146393776, 0.136819497, -0.161653802, 0.202596903, -0.184190035, -0.143676028, 0.129627481, -0.0586775057, -0.181300387, -0.0238430016, -0.189769417, -0.0744324401, -0.197278708, 0.164129451, 0.0219707415, 0.0293897092, 0.0587765612, 0.0964035615, 0.15167059, -0.125168294, -0.190928459, -0.112992272, 0.0658306628, -0.0772390664, -0.199625686, 0.125136733, 0.016112512, 0.0507222563, -0.0624214858, -0.16135475, 0.0569047816, -0.0239417739, -0.0304762162, -0.194920689, -0.12425144, 0.00409839163, 0.107493088, -0.208759293, -0.066616863, -0.172572762, -0.0572636537, -0.0250401981, -0.186279193, 0.0375845768, 0.201264232, 0.04939197, 0.123899333, -0.155704662, 0.0954312757, -0.150194436, -0.055589918, -0.14039661, 0.131468296, 0.194920346, -0.212645948, 0.0513700098, -0.117145963, -0.108924069, -0.186193109, -0.0858286917, -0.074252367, -0.052907601, -0.174557745, 0.0896119028, -0.119890451, -0.0677545518, 0.141775265, 0.183063552, -0.098954916, -0.143848076, -0.180254698, 0.0703581721, -0.000212103128, -0.0897746533, 0.183473036, -0.0284350216, 0.0284716189, -0.0381336361, -0.20608604, 0.169497326, -0.0935021788, -0.162120327, 0.0298986882, -0.152690023, -0.0220084935, 0.0699769109, 0.09413068, -0.161180288, 0.107032284, 0.170551285, 0.0715923756, 0.0323232859, 0.098411873, 0.14979668, 0.1879002, -0.0492424816, 0.119373843, 0.0076083988, -0.0622389913, 0.184939489, 0.085078761, -0.205675215, 0.0704781264, -0.108920917, 0.160283193, -0.135330096, -0.0439995378, -0.0609262735, -0.146751195, -0.0557816476, 0.187445238, 0.112474993, 0.108281776, -0.1571922, -0.0101753175, 0.032023266, 0.0926543921, -0.0471730232, 0.121487752, -0.0342903174, -0.0375407673, -0.0172177386, 0.241554603, 0.127430961, -0.0501674153, -0.136261061, 0.0438360311, 0.275473982, -0.0898060501, -0.00404814957, 0.150418699, 0.26817739, 0.0120358318, 0.0627415776, -0.217566565, 0.0120521989, 0.231260166, 0.174179092, 0.20312205, -0.099578023, 0.131383866, 0.0526953712, -0.0166083407, -0.179985553, -0.0176230427, -0.16833955, 0.055621013, 0.16548951, -0.078905493, -0.102710724, -0.144292682, 0.193504497, -0.167036876, 0.143709898, -0.106144384, -0.158193961, 0.180407584, 0.134830743, 0.0780916661, 0.21605663, -0.203453779, 0.153617635, -0.0991857052, -0.259447694, -0.157837898, -0.0765701681, -0.166750148, 0.0323081128, 0.0766944364, 0.231664136, 0.099929817, 0.225088254, 0.0904840156, -0.0980547816, -0.139175221, -0.0406756736, -0.0503455848, 0.013110226, -0.236767709, 0.108082667, 0.0616400279, 0.12457861, -0.0175604355, 0.0778381824, 0.0382082202, 0.210355639, 0.0954632461, 0.211079672, -0.10271854, 0.0311335325, -0.0154708745, -0.20266667, -0.0589585006, -0.15951401, -0.0808824971, -0.206491053, -0.0773185492, 0.0643220842, 0.269766062, -0.0534514859, -0.0768430829, -0.181922227, -0.12921229, 0.0590348989, -0.0676625296, -0.163617879, -0.210261837, -0.108614251, 0.141992033, 0.292766303, -0.00388330221, -0.0342260152, -0.278354913, 0.202880338, 0.114471421, -0.0569821373, 0.209743157, -0.197622269, 0.11517106, -0.282697707, -0.177471429, -0.0363213867, 0.0715632513, 0.0966505781, 0.156586885, 0.00711535243, 0.193091586, 0.319586277, -0.077367425, 0.194643721, 0.133760348, 0.162715733, -0.213925645, 0.0577851124, -0.115082778, 0.0244967844, -0.233547971, 0.16115953, 0.116338134, -0.0176728424, 0.103588142, -0.0136159752, -0.0320229046, 0.0752808824, -0.0454647131, 0.141926035, -0.157470793, 0.0646567643, 0.116127677, -0.0982909575, 0.0018835736, -0.206134573, 0.0186304394, 0.119598277, -0.114110075, -0.196623132, -0.202344328, -0.0913590342, -0.201012149, -0.0851496235, -0.0685937256, -0.235107616, -0.12301024, 0.124149792, 0.0983350128, 0.0774306282, 0.0723523647, -0.215187356, 0.111336991, 0.127059489, -0.112067282, -0.00816392899, 0.126290902, 0.0156315081, 0.0512061268, -0.210605562, -0.0202413108, -0.145583779, 0.00709361816, -0.124394178, 0.180435747, 0.104641557, 0.0187026784, 0.0350805745, -0.163335904, 0.194162667, -0.0241593253, 0.117580511, -0.171764538, 0.225402132, -0.0720629022, 0.0310874283, 0.0749795213, -0.205305517, 0.124029838, 0.0928468481, 0.104787186, 0.122945972, 0.0687557608, 0.197842777, -0.038209822, 0.209728137, 0.148183659, -0.0895242766, 0.102743544, 0.158801213, -0.0225127339, 0.176194936, 0.0220577177, -0.0678962469, -0.0967836902, -0.167863473, 0.179799557, 0.148632124, 0.0381179079, 0.208649412, 0.0900598094, 0.143464074, -0.0833160579, 0.129522786, -0.0478451103, -0.0691998526, 0.0784664005, -0.0541049801, -0.142444491, 0.157873392, -0.0442984365, -0.0314130932, -0.0341217779, -0.190294713, -0.0624290369, -0.0108193904, -0.0722554624, 0.0450399257, 0.184874624, 0.0353574604, 0.250395238, -0.211719662, -0.0713019222, -0.0945236161, 0.0628559738, 0.113878533, -0.166120961, 0.0611039735, -0.0665954202, -0.190605044, 0.104317546, -0.00670157606, 0.197475791, -0.157059222, 0.0666453913, 0.190627366, 0.00203674077, -0.0640138537, 0.169015393, 0.158805847, 0.00249635987, 0.175454721, -0.11453028, -0.0718963668, 0.0581686459, 0.0863645673, 0.254797548, -0.0167599767, 0.0753724277, -0.191692099, -0.037594419, 0.0371002257, -0.0114472676, -0.129038393, 0.135102063, -0.0811199322, -0.0868073627, -0.140736476, 0.270534247, 0.211350933, -0.0777289495, 0.0280433893, 0.0301295258, -0.138493523, -0.226183578, -0.00809103157, -0.048917044, 0.134023279, -0.111272015, -0.131809756, 0.167289764, -0.0939597264, -0.0454141498, -0.199593216, -0.0715295821, 0.16763784, 0.155164659, 0.0330340266, -0.0935863256, 0.074379988, -0.055489637, 0.0121996375, 0.216600537, 0.0732028931, 0.106504105, -0.179512233, -0.0358368456, -0.192034081, -0.0353995189, -0.0244174004, 0.0996022075, -0.0177846104, 0.219992995, -0.101739459, -0.0576194376, -0.169102862, -0.0963000655, 0.0924205929, 0.0396039449, 0.0483620577, -0.0561504178, -0.0868818238, 0.0164745953, 0.0548049062, 0.114303872, 0.013754636, -0.0567086786, 0.102405623, -0.0438192934, -0.0643145293, -0.0401981324, 0.00962526165, 0.195387542, -0.162058115, -0.118062168, 0.0846031681, 0.0343922898, 0.0729532316, 0.186529264, 0.0633441284, -0.0136433439, -0.0180960745, -0.022626821, 0.130006075, 0.141576752, 0.0769681633, 0.0622897595, -0.126342788, 0.0708925575, 0.0250345729, 0.00250566704, 0.137845576, -0.0369660184, -0.186658204, 0.0200903825, -0.0130848829, -0.10494981, -0.0606996045, 0.169031233, 0.125592455, -0.081215255, -0.0654265434, 0.0523951836, -0.142207876, 0.254872948, -0.153936654, -0.188501954, -0.160121426, -0.134948, 0.205956161, 0.190052256, 0.16584532, 0.151236117, 0.0718697757, -0.080587402, 0.110667244, 0.0943986848, 0.181700706, -0.00617637718, -0.208006665, 0.14149186, 0.0434235521, -0.0528380871, 0.0149466833, -0.00435288716, 0.181254312, 0.10414812, 0.132486179, -0.0475688763, -0.139805526, 0.061016947, 0.088329263, 0.104247503, 0.237457544, 0.22448419, -0.0426649414, -0.0163636543, -0.204058439, 0.163758263, 0.243123114, 0.234052137, 0.0471326299, -0.117478944, -0.0863664374, 0.0787322223, -0.159595221, -0.173156038, -0.0570174493, 0.086930953, -0.141002566, 0.124750815, 0.191485867, -0.202254176, 0.205454722, 0.166258335, 0.0726499707, 0.0952544957, 0.100071169, -0.202629045, -0.172590211, -0.13892965, 0.0231076777, 0.111921228, 0.274842918, 0.0941486955, 0.0641628727, -0.142406732, 0.0568496808, -0.0287323724, 0.0187774654, -0.0521207936, -0.164493352, 0.131963298, -0.0280933343, -0.212045416, -0.104063354, -0.0864547491, -0.204800725, -0.0237307753, 0.0920451134, -0.0136097614, -0.11391791, -0.264806271, -0.201454163, 0.147936925, -0.146814078, 0.171959713, -0.124607295, 0.129478768, -0.204661041, -0.0736282244, 0.190738454, 0.0476327986, -0.0412670225, 0.103763528, -0.215454429, -0.0301665645, 0.00799800269, 0.193996519, 0.155501172, 0.0539092608, 0.0650432557, 0.226527035, 0.180688441, -0.182288006, 0.0930174738, 0.260853142, 0.016753193, -0.214730203, 0.0154327303, -0.0481189452, 0.0598105043, 0.0232905801, 0.130197376, 0.17757155, 0.0245893449, 0.151050985, -0.107956119, -0.240185767, 0.00206723274, -0.0504090339, 0.212470889, -0.160272613, 0.239395365, 0.203135297, 0.189087495, 0.0853048265, 0.171777859, -0.029955145, 0.11319828, 0.0216485877, 0.00814698357, -0.110079348, 0.0574759692, -0.0117787374, 0.0587957054, -0.0188551173, 0.187958941, 0.201361075, -0.212008983, -0.150154889, -0.0777181834, -0.0097771734, 0.262629092, -0.0380698293, 0.043783132, 0.22858268, -0.0257687774, -0.0354431905, -0.0717736334, -0.0261267014, 0.238806605, -0.0407217331, 0.00614640862, -0.00211061444, -0.158218428, -0.0143331885, 0.0456409603, -0.0461011529, -0.145143121, -0.0836481154, 0.0455304757, -0.164061174, 0.137408197, 0.160984814, -0.05268538, 0.0676740408, 0.082190454, 0.213888645, 0.108864151, -0.229466036, -0.00585621083, 0.220650971, 0.128265545, -0.0412900858, -0.21077244, 0.15473862, -0.119168244, 0.1800441, 0.207246855, -0.11915756, -0.0156303793, -0.198259041, 0.0665771812, 0.108989105, -0.00986023247, 0.165291443, 0.0965227336, 0.00951856375, 0.0554960519, 0.0457220227, 0.196098253, 0.128513381, 0.0316233784, 0.00890362263, 0.166757986, -0.0175813287, -0.158623844, -0.20614323, -0.167428017, 0.00473146141, -0.106193721, 0.15801324, 0.00607329607, -0.00859092176, -0.154501185, 0.0736638755, -0.172929317, 0.178296432, -0.204777554, -0.0184551328, 0.0859390348, -0.0314055979, -0.110383652, 0.024170354, 0.0688661188, 0.103539482, 0.1746995, -0.0174282789, -0.188645795, 0.130957142, 0.161050007, -0.171988711, -0.124570034, 0.18495886, -0.173855573, -0.0370936096, -0.142793447, -0.145858899, 0.182163581, -0.183721334, 0.0315484852, -0.0502992272, -0.0749663711, -0.187164277, -0.0742956847, -0.130046368, 0.0317636281, 0.142129526, 0.0862586349, 0.0828672573, 0.0140935238, -0.079975754, 0.173597023, 0.141604081, -0.0771767423, 0.118548639, 0.0442024469, 0.0727466717, 0.266035914, -0.00593646383, 0.260059625, 0.144515678, -0.0130532747, 0.188891038, -0.0634195805, -0.0261913594, -0.0180802289, 0.237168074, 0.171025172, -0.130810335, 0.208993554, -0.030096842, 0.0740133673, 0.241876543, -0.184140071, -0.0688809901, -0.146465331, 0.16539228, 0.190757021, 0.17606993, 0.196502313, 0.136242479, -0.0804710537, -0.00782729965, 0.188913107, -0.0548046194, -0.0303347055, 0.142485619, 0.151637778, -0.158051103, -0.0266635474, 0.0728768855, 0.137775302, 0.125231311, 0.0346932858, 0.163109958, -0.205083966, 0.0756561756, -0.116977692, 0.0437464379, 0.231042966, 0.193829939, -0.18651934, 0.149564371, 0.154574603, -0.0290720891, -0.0690897927, 0.179843798, -0.0955478922, -0.0206622425, 0.190791145, -0.122945897, 0.125592127, 0.00321447477, -0.195028916, 0.0442178249, -0.104046471, 0.0260952171, -0.0816862285, -0.110913567, 0.091348283, -0.115662403, 0.251517475, -0.21434246, 0.175582513, -0.14993903, -0.0990529507, 0.0514201038, 0.150468886, 0.228353143, -0.173500925, -0.00461063208, -0.0714868903, 0.143813297, 0.217226163, 0.114283666, -0.197505504, 0.0496195182, 0.0727943853, -0.0745235234, -0.0619089901, 0.0918129012, -0.117093414, 0.0321687013, 0.236869738, 0.126950324, -0.162127212, -0.119039662, 0.161647394, 0.231011108, 0.177849144, 0.147918016, 0.133619756, 0.190788567, 0.0492400676, -0.00180678465, 0.0893449634, -0.148697823, 0.177664801, -0.0726399198, -0.0793330893, -0.225488186, 0.131051272, -0.113395549, -0.14153862, 0.0294948965, 0.191074476, -0.00509508047, -0.0429674871, 0.0682959855, -0.122674003, -0.110053435, -0.0392141566, 0.0516043007, -0.0405695885, 0.278859168, 0.146024361, 0.223367631, 0.179515615, 0.182836056, 0.0309408158, 0.0159752686, 0.00173792825, 0.11343246, -0.10914018, -0.056721732, 0.0177230816, 0.175182432, -0.036981035, -0.131743401, 0.207399696, -0.0125906104, 0.192897528, 0.10380502, -0.128706738, 0.141425639, -0.141085252, 0.0864470005, -0.00618862314, -0.00134076655, 0.00479231775, -0.11014533, -0.135056555, 0.00566653907, -0.179885507, 0.197231576, -0.0278437734, 0.132824823, 0.150243133, 0.151170567, -0.0333556682, -0.0339126848, 0.0283680595, -0.025435755, -0.0908457041, 0.0670256168, 0.119782694, -0.048878938, 0.0382228903, -0.106433287, -0.129820496, 0.0346301049, 0.0843395144, 0.0345586091, 0.151655838, -0.0818703771, -0.081794247, 0.115935832, -0.0413574092, -0.00304169138, 0.0973383635, -0.00981269684, 0.0169961806, -0.168726087, 0.124752775, 0.0624595955, -0.166663989, 0.134228542, -0.133986801, -0.117507249, -0.183109924, -0.0409472734, 0.190115988, 0.0337236971, 0.117162749, -0.076600574, 0.129812434, 0.134825528, 0.0260062516, 0.0371112674, 0.177381799, 0.183222786, 0.216518879, 0.015962854, 0.0845715106, 0.108023062, 0.135057315, 0.000637001474, -0.203383252, 0.196280256, 0.0818561018, -0.100496322, 0.158635378, 0.179170743, -0.0156604201, 0.093567811, -0.101123378, 0.00368472934, 0.0540641397, 0.180312157, -0.201012507, -0.00493814051, 0.0403486565, 0.10555122, -0.219209358, -0.0529356785, -0.0400650203, 0.158233479, 0.10751909, 0.123106666, -0.0264859833, 0.143902779, -0.155771375, -0.109103367, -0.0625805184, -0.0451420695, 0.210679486, -0.194820687, 0.07988628, -0.162504762, 0.208094731, -0.150656149, -0.078792125, -0.12391606, 0.0141808093, 0.172131687, -0.108649395, -0.0934482217, -0.219430164, 0.193088472, 0.0839586705, -0.0547866635, 0.0759218782, -0.0979883671, -0.0717851892, -0.133541152, -0.214100048, -0.147924244, -0.00851948559, -0.0822613388, 0.111076437, 0.204227194, -0.0590670258, -0.0866161436, -0.0972947702, 0.0178795159, 0.0895289332, -0.0690636188, -0.0857937858, 0.16783753, -0.0259044375, 0.00509806909, -0.225554511, 0.154907301, -0.146912664, 0.268833876, 0.140848532, -0.159942165, 0.204923227, -0.16968435, -0.0109424917, -0.140655488, 0.00905802846, 0.0975849852, -0.113203347, -0.00286432612, -0.00585176935, -0.163264215, 0.177411392, -0.200985014, 0.00323767564, 0.0647737458, 0.0477584526, 0.103176244, -0.0821804181, 0.0348460563, -0.110611327, 0.148955032, 0.269896477, 0.0960517451, -0.103157543, -0.162139267, -0.149393424, 0.125260234, 0.070246011, -0.225312755, 0.25742054, -0.0397864655, 0.177335784, -0.0546780899, 0.248964921, -0.166126356, 0.192700773, -0.00790695101, -0.0664229989, -0.153038487, -0.129117221, -0.0757997856, 0.0386017896, -0.135388434, -0.158859819, -0.104986891, 0.146457687, 0.199433178, 0.066154249, -0.27667287, -0.118511088, -0.0179567039, 0.222479478, 0.0455367491, 0.243386254, -0.120252974, 0.132388383, 0.00776485447, -0.194177583, -0.0780516565, 0.00999934599, 0.11524263, 0.142233551, -0.0642258972, 0.186899021, -0.103108883, 0.099964574, 0.237639084, 0.121256396, 0.0142423958, 0.202542499, 0.20030944, 0.180703923, -0.214075804, 0.0230388809, -0.299164712, -0.128671005, -0.189861313, -0.167792231, 0.0813844353, 0.00933712721, 0.0428303629, -0.1023985, 0.174391836, 0.253679901, -0.0937102586, 0.0857886672, -0.158551842, -0.167360649, -0.0763060898, -0.0540213883, 0.133122638, 0.148575723, 0.0668005571, 0.152676195, -0.0732476413, 0.0157247335, -0.270311266, -0.0190660674, 0.212057456, 0.182492748, -0.241901889, -0.0313768871, 0.228386506, 0.0656861812, 0.192671508, -0.157984391, 0.0745935887, -0.0429898053, -0.122312985, 0.124423012, 0.0292300582, 0.181159899, -0.110646807, 0.205835596, -0.127989545, 0.139688984, 0.0181228518, -0.0549869686, -0.161712885, -0.0697539151, -0.0804900229, -0.0285761952, 0.123424694, -0.207021698, 0.0395707637, -0.211159229, -0.045374617, -0.150724575, 0.179440662, 0.103816822, 0.015124768, 0.0048571527, -0.185660616, 0.0693678111, 0.0240155458, 0.0238517523, -0.130017757, -0.210529521, 0.112137035, 0.178406164, 0.19203876, 0.21485664, 0.191359922, 0.0654983968, 0.166367605, -0.0858131945, 0.0867324322, -0.141689003, -0.137133151, -0.210735589, 0.216141865, 0.00645007193, -0.170115247, 0.0192143917, 0.156424567, -0.12158598, -0.170511737, 0.118564084, -0.203893989, -0.100373045, 0.206237301, 0.0579547733, -0.109020285, -0.159191296, -0.196344331, -0.10288664, -0.0650167316, 0.0364720076, 0.210455045, -0.198279276, 0.0561158136, -0.191313118, 0.021069834, -0.0339165032, -0.191652551, 0.198695317, -0.120528094, -0.0548847243, 0.0808626562, -0.00428579329, -0.102671824, 0.117770836, 0.140487507, 0.134317502, 0.156712055, -0.212678373, 0.115886249, -0.0798269957, 0.215774462, -0.161133751, 0.178629026, 0.0955588222, 0.155450925, 0.0492355675, 0.135866612, 0.202169314, 0.0468329042, -0.150953293, -0.0446973443, 0.103053465, 0.0478212684, 0.214107037, 0.135672152, 0.200946644, -0.174147338, 0.12126869, -0.139116272, -0.0563006103, 0.0277512744, 0.246417493, 0.0611405782, -0.0119189397, 0.208439246, -0.0356294885, -0.170967788, -0.115360253, -0.129960269, 0.144377574, 0.0454087257, 0.259763271, -0.105527014, 0.055321455, -0.0526598319, 0.159842834, -0.0482077226, 0.236779749, -0.132585362, 0.189681903, -0.0961048529, 0.0563793406, 0.18519479, -0.127709776, -0.0987681523, -0.0303634182, -0.0687099472, 0.0578852296, -0.0381461047, -0.18619667, 0.12401966, -0.121132657, 0.225062236, -0.205080852, 0.0551929399, -0.0777834952, -0.053174451, -0.199143633, 0.159538761, -0.238657549, 0.220129281, -0.114376858, 0.221257493, -0.255461693, 0.0300092585, -0.0607489645, 0.126692057, -0.112293094, -0.0986434072, 0.0438456684, -0.130739585, 0.0128232781, 0.166859791, 0.0306993425, -0.0176246464, -0.130978495, -0.0725799501, -0.00697065098, 0.149285182, 0.0522971042, 0.0522838607, 0.132519081, 0.192778155, -0.0416352339, 0.109511234, 0.202514991, -0.189964101, 0.0592628978, -0.133078381, 0.249684885, 0.151773691, -0.0527177453, -0.100954384, 0.124180362, -0.203475311, -0.118713893, -0.0816718787, -0.0157442, 0.100288361, 0.124790654, -0.027971575, 0.0515414514, -0.152316317, -0.139562219, -0.135580957, -0.084609136, 0.167367682, -0.169176459, -0.128676862, 0.160356179, 0.167749211, 0.208847791, 0.059897989, 0.161345467, 0.195118994, 0.11026185, -0.0473038405, -0.162515476, -0.140200004, -0.138756335, -0.189846769, 0.20646067, 0.0327555984, -0.222942144, -0.0198731795, 0.0467148684, 0.0791418999, 0.0614629388, -0.126075357, 0.108883843, 0.00917934161, 0.0830445662, 0.080400981, 0.113189146, -0.147388667, 0.200981006, 0.09387137, 0.0662245005, -0.127312094, 0.101593748, 0.146900043, 0.230416954, -0.221930906, -0.0331053957, 0.17240724, -0.0221072081, -0.0760479346, -0.20360899, 0.112684511, -0.138931423, -0.162155733, -0.119198255, -0.126619726, 0.012630037, -0.109421387, -0.166782975, -0.182280928, -0.172797754, -0.0645593479, 0.0926890373, 0.0646796972, -0.123785369, 0.259334207, -0.0265048742, 0.0963960364, 0.0207417514, -0.0640984923, -0.0827390105, -0.134210065, -0.0423009247, -0.0835836828, 0.077250883, 0.0914835781, -0.000481657393, 0.0296047516, 0.176210508, 0.155236304, -0.120164134, -0.0224553142, 0.136641458, 0.0316355117, -0.099346526, 0.0761687532, -0.172814578, -0.228517711, 0.158629566, 0.0357749611, 0.00243570539, -0.0157305691, 0.0191846807, 0.00691910414, 0.0227921773, -0.0236533042, -0.18064791, 0.00115233322, -0.156837761, 0.111577243, -0.148221925, 0.230223015, 0.0173706133, 0.206947878, -0.0331011862, -0.160140678, -0.0975864902, -0.116723441, -0.13038072, -0.0243134685, 0.12657474, -0.0980337113, 0.175942108, 0.00192179182, 0.0473435558, 0.205429345, -0.0407878272, -0.213827103, 0.10833922, -0.0446451604, 0.0655935183, -0.188038319, -0.00301687419, 0.0675255656, -0.143765509, 0.00169246364, -0.0247743782, 0.065864265, -0.127450123, 0.186487421, -0.184591785, 0.0808997974, 0.0317924172, 0.00249277428, 0.0951853916, 0.276850134, 0.122914597, 0.0458479226, -0.112578034, 0.171549395, -0.214462727, -0.219333857, 0.215502247, 0.0376836024, -0.101821326, 0.23026073, 0.149181589, -0.116133168, -0.0090032015, -0.116861179, 0.256513149, -0.162931934, -0.112243503, 0.00128614902, 0.0244441722, -0.213078201, -0.0275032464, 0.0797179267, 0.111045495, 0.246224776, 0.0375076756, -0.0120324278, 0.122870028, 0.260363281, -0.0590779483, 0.0948166922, 0.153928548, -0.166328102, -0.198541239, 0.0432137474, 0.0723608881, 0.0856808871, -0.0166272782, 0.121594638, -0.196286201, 0.0552772507, -0.0785965696, -0.0785046741, -0.0733379275, 0.0284803696, 0.183244765, -0.0545121506, 0.183057174, 0.0930560529, -0.0827762261, -0.214541987, 0.0781526715, 0.0538695231, 0.179998606, 0.187902153, 0.0758102015, -0.117636815, 0.0950077325, 0.158064738, 0.0105737597, 0.0903970301, 0.108313836, 0.15097709, -0.0819445699, 0.0761458278, -0.140456557, 0.131802991, 0.0474786013, 0.155419514, 0.0239446163, -0.0219119042, -0.135106996, -0.144528925, 0.202310726, 0.0346909016, -0.190453961, 0.0817741007, -0.110087767, 0.0702924579, -0.0885792077, 0.0543277413, -0.0371818244, 0.1415499, 0.0944445878, 0.0789010972, -0.0174358636, -0.187914088, -0.0285935998, 0.206651524, 0.162923053, -0.0869459808, -0.17593582, -0.0593883246, 0.12480326, -0.130898282, -0.130268216, 0.0238823146, -0.129311413, -0.167941093, 0.0979045182, 0.115539357, -0.0248285532, -0.0738229454, -0.0171255767, 0.214699998, -0.214020938, 0.140577748, -0.122401878, -0.0789570361, -0.0618365258, -0.0654320568, 0.0157889575, -0.0293144584, -0.185034052, 0.036581561, 0.194275334, 0.1666383, 0.215620413, -0.100140139, -0.0502271801, 0.148168072, 0.105212435, 0.172577128, -0.205824286, 0.108652189, 0.156266138, 0.0341610163, -0.207641378, 0.0638252646, -0.162136316, 0.0771442205, -0.136415035, -0.0285003185, -0.0351519659, 0.0870053843, -0.13288036, 0.0186352301, 0.0405196398, -0.0903854445, 0.0850627348, -0.0760384947, -0.237707302, 0.177195832, 0.128395244, 0.0780189186, -0.200771526, -0.0849047601, 0.0701752678, 0.260807902, 0.156773731, 0.19866395, 0.0359680429, 0.0136158485, -0.113989539, 0.0786288232, 0.202783525, -0.145905748, 0.0732347518, -0.0434487239, 0.204440325, -0.00198599696, -0.118598729, 0.0120036881, 0.201528028, 0.209207103, -0.0491646491, 0.15841648, 0.136860237, 0.0266900212, 0.0796270967, -0.100128114, -0.114517465, -0.0816531703, 0.195008367, -0.0176160038, 0.113583505, -0.074151665, 0.154809341, -0.0299604684, -0.128933713, -0.00159797072, -0.211855963, -0.238786757, 0.0815278813, 0.179436997, 0.165538907, -0.105617143, 0.0446293801, -0.116550677, 0.212327167, -0.186529025, 0.178048402, -0.152893737, 0.211425483, -0.0932270586, 0.134178355, -0.082460545];
    bias_6 : ARRAY[0..63] OF REAL := [0.0747542903, 0.0747530833, -0.00429329416, -0.0110996887, 0, -0.0352521576, 0.0479723401, 0.0685250089, -0.0227601323, -0.00580839999, 0.0100521399, -0.0113847172, -0.0245158654, 0, -0.0200175196, 0.0475497283, 0.0741227865, -0.0268050022, -0.053697817, -0.00196474558, -0.0566426925, 0.0682095364, -0.00484778127, -0.00283427443, 0, -0.0188507643, 0.0644902736, 0, 0, 0.00199445919, 0, -0.00884012785, -0.00463645626, 0.0127481027, -0.0124424472, -0.047869388, -0.0151582286, -0.0145472726, -0.0152692702, 0.107757747, -0.032102257, -0.00659875572, -0.0174676776, -0.0266960394, 0.0917816684, -0.00874918327, 0, -0.0106172459, -0.0176149886, -0.026105281, 0.0043185926, -0.0422325172, 0.00292709749, 0.00419008406, 0, 0.0809127167, 0.0434060618, -0.00947956275, -0.00768119283, 0.0844815671, -0.00330898049, -0.0406921245, 0, 0.0103572262];

    weights_7 : ARRAY[0..4095] OF REAL := [0.0985890701, 0.261478722, -0.0590967536, 0.0771033317, -0.00640187413, -0.0827855617, -0.230103448, 0.0237006657, 0.211521849, -0.133053824, 0.144778341, 0.0126608955, -0.264563471, -0.0297934134, -0.171915665, -0.144233555, 0.184128761, -0.199485853, -0.128364205, -0.10924013, -0.0942144915, 0.12244907, -0.134638637, 0.159754649, 0.102856718, 0.193186775, 0.0345768109, 0.0443875194, -0.0223890841, -0.0877400488, -0.224890769, -0.0661405474, -0.0205741599, -0.132689729, -0.134608626, 0.0912717804, -0.0320888869, 0.207671627, 0.0316983312, -0.263397604, -0.159447983, -0.123716153, -0.0258523077, 0.231007561, -0.107568942, 0.228946403, 0.115262851, 0.202499971, -0.222295597, -0.0375091396, -0.23364678, -0.123035237, -0.0525233448, -0.0821483433, -0.12599954, -0.358725101, -0.0378492288, 0.14551425, -0.117850862, 0.0302092116, 0.136658132, 0.0596454889, 0.0601940267, -0.115125708, 0.190094337, -0.0647920668, -0.120055743, 0.00146726007, -0.178027615, 0.0304296073, 0.155361906, -0.165448382, -0.0763782412, -0.227639481, -0.156574205, 0.134376928, -0.335413128, -0.213705391, -0.0161788668, 0.176306963, -0.0786898807, 0.0378909893, -0.156903595, 0.0734621733, 0.145642534, -0.0653213263, 0.00195453106, -0.167763978, -0.112661101, 0.116725579, 0.228570595, 0.185373247, -0.0674858838, 0.123988092, 0.114007965, -0.0454010144, -0.077554442, -0.0201824624, -0.275262088, -0.114391603, -0.0663379133, 0.280113071, -0.112193778, 0.0486323275, -0.137166336, -0.0401128717, 0.0894181207, 0.00908427685, 0.179754227, -0.0671511367, -0.120330289, 0.114102527, -0.226583004, -0.0849781409, -0.0418890789, 0.17914106, 0.204921558, 0.0455944687, -0.0450889394, -0.0856394097, -0.113558985, 0.166775107, 0.0186151415, 0.211812183, 0.186384693, -0.132189557, -0.156687155, 0.191395983, 0.110498078, 0.139661208, -0.0920242742, 0.222033158, -0.00120364304, 0.00128853915, -0.0888353512, 0.211148933, 0.0156825483, 0.197753608, -0.181704342, -0.159737736, -0.0235950705, -0.0353642218, -0.00933676027, 0.126852483, 0.171151608, -0.0931896344, -0.0475037992, 0.138531879, -0.194260553, 0.0657681227, 0.136853874, 0.0619690791, 0.100470409, 0.0687212795, 0.0456814691, -0.0741193444, 0.143832967, -0.0251761973, -0.0440490879, -0.197995454, -0.100512169, 0.0636347532, 0.194363266, 0.14988251, 0.117436595, 0.0813431665, -0.0845726654, 0.041465167, -0.143196225, -0.13916254, 0.0370236412, 0.106373869, 0.133378014, -0.0168813877, 0.0678688437, -0.0221709907, -0.178990752, -0.0615577288, 0.208223164, 0.117776372, 0.0550451688, -0.11717312, -0.106960475, -0.132753909, 0.0749269575, 0.0704251528, -0.121250421, -0.182553753, 0.0348108932, -0.169337317, -0.0431644917, -0.06188545, -0.044683557, 0.0603879951, -0.086644128, -0.0278274007, 0.146163434, -0.0545757636, 0.0299487282, 0.174511701, -0.0916855708, -0.153672263, -0.0549600422, 0.0154589014, 0.00445316266, -0.102152765, 0.0601579957, 0.166933239, 0.040345829, 0.268830568, 0.154072955, 0.10402365, 0.0998772457, 0.0329706669, -0.18961744, 0.16987507, 0.083305344, -0.127246037, -0.209014222, -0.192148447, -0.160925955, 0.114261568, -0.133135706, 0.0742198899, 0.115098283, 0.229157656, 0.0866794065, -0.141607061, -0.00846149493, 0.1364851, 0.165410504, 0.177613571, -0.198162705, 0.204134092, -0.171739325, -0.204839557, 0.274487436, -0.0561079755, -0.183752149, -0.0607956015, 0.128661469, 0.0149638271, 0.00135228958, 0.187765002, 0.0477933511, -0.146877944, 0.164612621, 0.104129799, 0.0751872286, 0.09320952, 0.17067422, -0.122773752, -0.0966985524, 0.148433819, 0.166774407, -0.050018996, 0.107592955, 0.17758055, -0.0572009236, -0.115987271, 0.10496451, 0.0970115513, -0.0402181149, 0.143645063, -0.114797451, -0.0233546644, -0.0524974316, -0.180076912, 0.134013399, -0.138859093, 0.0046711117, 0.0682574362, -0.11045447, 0.101280972, -0.141288802, 0.131182745, -0.104055196, 0.1359476, -0.105594479, -0.199489638, -0.100357562, -0.184324607, 0.0823699385, 0.111964449, -0.0532657355, 0.0663902014, 0.177432373, 0.210205242, -0.210125804, -0.0332980007, 0.096206829, -0.0193504691, 0.167757437, 0.0213211328, -0.105646975, -0.073984772, 0.203198329, 0.0314622223, -0.175412863, -0.122094072, 0.0986203104, -0.122762077, 0.19236134, 0.135295138, 0.182322904, -0.103380427, 0.144614473, 0.0554241389, -0.175479814, -0.0391083062, 0.191711053, 0.121323869, 0.115582779, 0.181385979, -0.192489818, -0.173019394, -0.173292458, 0.0201414824, -0.0125766397, -0.0790846944, 0.0685555041, 0.167224765, 0.189211607, 0.210358679, -0.0415095538, 0.126387641, -0.0842779204, 0.0439397581, 0.00644816831, -0.152137846, -0.152992308, 0.0245475248, 0.192403287, 0.163964272, 0.116401248, 0.0257411487, -0.142266706, -0.146128058, 0.0102699744, -0.0180726349, 0.197232619, 0.193206668, -0.0754495487, 0.134801105, -0.00232620165, 0.225295782, 0.0273058284, -0.154496655, -0.201236218, -0.157684937, 0.187730253, 0.115707032, 0.131131858, -0.167114601, 0.047023993, -0.0567260347, -0.0668960586, -0.083985351, 0.0849857107, 0.0702214763, -0.179636031, -0.0277230721, 0.162856936, -0.20755665, 0.160055265, -0.182279021, -0.235589236, -0.151465133, 0.0571531281, -0.148302287, 0.248307049, -0.12540251, 0.115537778, -0.190976933, -0.0118816132, -0.0110264076, 0.138518065, -0.122859232, -0.0116230948, -0.185463518, -0.193349451, -0.160361007, 0.130532175, 0.209439963, 0.0375103466, 0.285149574, -0.158949748, -0.277013332, 0.153673515, -0.260961682, -0.172621742, 0.167940751, 0.207475811, -0.175017715, 0.145652935, -0.026749935, -0.0299806502, -0.266049534, -0.196326286, 0.033781562, -0.0726778582, -0.262074381, -0.0483580381, -0.143439263, 0.141321659, -0.00700642727, 0.292194456, 0.185188755, -0.0455660783, 0.101106308, -0.0083050346, 0.150430575, 0.15473111, 0.277323723, 0.112545229, -0.0247835293, -0.176015452, -0.04111927, -0.0102430824, 0.111235037, 0.142509177, 0.131318763, -0.15878965, -0.124645673, 0.191819474, -0.0986970142, 0.120010592, 0.279321134, 0.121246748, 0.170530006, 0.0124538634, 0.146209851, -0.0564521439, -0.453932881, -0.115464613, 0.0486782379, -0.212593615, 0.0844182074, 0.152913198, -0.0890955701, -0.014261798, 0.0763275549, 0.094609946, 0.16527921, 0.152573839, 0.215471298, -0.189632729, 0.0542746969, 0.0475845337, 0.165836349, -0.248436794, -0.139802009, -0.117795072, 0.0680505931, 0.127019078, 0.141767994, 0.108608454, 0.0795560554, 0.215438023, 0.253515422, 0.0968242809, 0.0465329401, -0.0367862582, 0.205732152, 0.0410595387, 0.14549467, 0.0515940823, -0.204010546, 0.097479187, 0.136549056, -0.0882421583, -0.231916368, 0.0916896313, -0.097374104, 0.108968385, 0.064018704, 0.0505693108, 0.151754782, 0.0724061951, 0.0685940981, -0.0536143109, -0.00958465319, -0.0650544614, -0.118865497, 0.0617310181, 0.164938733, -0.125389904, -0.0580696389, 0.076752767, -0.0623037033, -0.0602061898, 0.14020063, -0.0644329116, 0.185091019, 0.00150486734, -0.0492826067, -0.230618313, -0.0963186398, -0.0396718048, 0.0157787632, 0.147863075, 0.136901587, -0.0209644865, -0.0838856548, -0.0987434536, -0.0661321655, 0.0437461026, -0.125251681, 0.245231941, -0.142143026, 0.178793207, -0.120658711, -0.252990127, -0.0960166603, -0.148348227, 0.217699945, -0.152953058, 0.0320299491, 0.0397147648, 0.20091784, -0.297417134, 0.043796204, 0.0147441905, 0.0458022691, -0.151441351, 0.0129484637, 0.0644230098, -0.122672424, 0.11798434, 0.212057024, -0.0869171694, -0.126012012, -0.04658252, -0.0954014957, -0.244200468, 0.145332858, 0.0195005015, 0.189192265, -0.230275482, -0.0202685073, -0.150195628, 0.13925834, -0.0658622757, 0.158107281, -0.0311671887, 0.00751672499, -0.177279904, -0.0161855966, -0.106229313, -0.159273162, -0.194914743, -0.1878708, 0.0287032183, 0.288048238, -0.0252802446, -0.0553182103, 0.14248237, -0.203866616, -0.238840014, -0.207598493, 0.112077221, -0.100770809, -0.0132202683, 0.131064698, -0.162306666, 0.10710378, -0.166209847, -0.00958471466, -0.105003767, 0.24485141, 0.152514249, 0.208566174, 0.162460268, 0.00807126984, -0.141904116, 0.108676672, 0.125443801, 0.036231447, 0.135343865, -0.187444642, 0.0880331844, 0.023205962, 0.00651972136, -0.00225225091, 0.183123365, -0.118129879, 0.130323112, 0.107369676, 0.211500779, -0.0843634605, -0.156388134, 0.207216874, -0.0687728524, 0.0857001096, 0.0248294771, -0.100912109, -0.157147497, 0.0598580688, 0.0957521722, 0.153322056, 0.0638879687, 0.0558222681, 0.13312462, 0.0504909046, 0.184043959, -0.147291183, -0.0967333466, -0.0938999057, 0.0367397517, 0.0814364702, -0.111346483, -0.120195106, -0.137015536, 0.00596247334, -0.127521366, -0.168997496, -0.0679924712, 0.0334541053, 0.0365803689, -0.0112984832, -0.0791522115, 0.165152445, -0.0490483344, 0.145707756, -0.203866005, -0.0773670673, 0.187672272, -0.124051414, 0.118377551, -0.152038693, 0.187986448, -0.178593695, -0.0927914903, 0.08069361, 0.205642715, -0.054671783, -0.0563890673, 0.062154606, 0.0556793362, -0.077488631, -0.237223327, -0.00743269641, 0.0303223412, 0.1891305, 0.115924723, 0.243285507, 0.128094137, 0.0924103409, -0.173196748, 0.186365053, -0.102543443, 0.0903031752, -0.0225095805, -0.0684509724, -0.0492378138, -0.142380729, 0.273817688, 0.162142336, 0.0942962393, -0.196417257, 0.0544637963, 0.0642177686, -0.0781479776, -0.00544341793, 0.0882533863, 0.135036305, 0.153385952, 0.060867317, 0.0675654262, -0.190924585, -0.0308644846, 0.209309757, 0.23535271, -0.114015281, 0.211691156, 0.103498377, 0.175216466, -0.0897360072, -0.178171828, 0.188865781, 0.184034958, 0.143535584, -0.0759150386, -0.144946337, 0.123703592, 0.072421141, -0.073435992, -0.120332345, -0.207936838, 0.0859730244, 0.089198038, 0.21525383, 0.042071078, -0.188023686, -0.222388178, 0.173431069, -0.0430555344, 0.15827693, 0.0902394876, 0.192961678, 0.073467873, -0.000299184467, -0.143207088, 0.194787577, -0.0937701017, 0.147017911, -0.167207763, 0.0221077409, -0.148127094, -0.0726192892, 0.0140165687, -0.131738737, -0.107379422, -0.0532393269, -0.183383986, -0.132864356, 0.14306511, 0.166543275, 0.0633267611, -0.00475004269, 0.159882694, 0.0209031757, 0.193773642, 0.0460488647, 0.00657480629, 0.135696039, -0.122650474, -0.0921338946, -0.0184501112, 0.197395191, 0.149274558, -0.212168857, -0.0961322784, -0.0972493216, 0.061156068, 0.0288367011, -0.129334092, -0.0287208185, -0.12547949, -0.109855622, 0.0713636428, -0.202687904, -0.0736791939, -0.170345217, 0.00483758748, -0.0566800907, -0.0133493776, 0.177170977, -0.16139634, 0.0383036919, 0.18136698, -0.0358033031, -0.158096969, 0.122688517, 0.081486389, 0.160581172, 0.210082605, 0.139138475, -0.0031660106, 0.0011371508, 0.153799191, -0.0630362555, -0.0959898457, -0.0677730069, 0.0763605982, -0.0591884851, -0.103758797, 0.0877787992, -0.203684002, -0.213626981, 0.216784999, 0.0821806788, 0.0854039118, -0.0622716844, 0.178851873, 0.0519754291, -0.102133691, -0.0585566014, 0.0188398492, 0.202151239, -0.104732491, 0.27045393, -0.0917108878, -0.208633393, 0.156232789, 0.231986329, 0.132011876, 0.000424101949, -0.220415235, 0.295938492, 0.0743808001, 0.14029865, 0.242455915, 0.23396118, -0.245414257, -0.195483923, -0.114712641, -0.0220132805, 0.322085798, -0.021815693, 0.282940984, 0.12972188, 0.131338835, 0.25256893, -0.182917267, -0.158058509, -0.129873797, 0.0281693563, -0.139118776, -0.060282778, -0.288214117, 0.18269442, 0.0694092885, 0.122847252, -0.0459760986, -0.18629986, -0.000292814599, 0.19988957, 0.157423139, 0.132337287, 0.124669015, 0.156890973, -0.164955139, -0.0223253407, 0.294166148, 0.301510572, 0.13682279, 0.0792005882, -0.100755952, 0.0107995598, 0.122480787, 0.0160061363, 0.146093562, 0.0933857411, -0.00256964564, 0.0729778558, -0.193990499, 0.00561368465, 0.168780282, -0.0343219191, -0.16398114, 0.19884105, -0.170096159, 0.0851236135, 0.046119079, 0.149938866, 0.106523618, 0.0622120649, 0.194288179, 0.153273478, 0.0731689781, 0.00548323989, 0.150967196, 0.0232321769, -0.163167983, 0.0613376349, 0.199462637, -0.0988652036, -0.202331737, -0.201972619, -0.0975645036, -0.103157334, -0.0671368837, 0.0251828581, -0.12365777, -0.0824821144, -0.0295259356, -0.200477883, 0.213229522, -0.126918197, -0.0524763167, -0.0709132403, 0.13771455, 0.182151392, 0.0844053477, 0.192415133, -0.0920736194, -0.0465842038, -0.146784067, -0.0747133791, 0.186533436, -0.201628059, 0.102212504, 0.176582918, 0.0926011056, -0.0415422022, -0.173487782, -0.145804495, 0.138758883, 0.215857342, 0.118435606, -0.183083788, -0.206599399, 0.0207605958, 0.0811169297, -0.150482222, -0.0474843644, 0.148732826, -0.0435940437, 0.168024451, -0.111467153, 0.138727993, 0.0159117766, -0.0708138347, -0.0325546637, -0.187760904, -0.0735307932, -0.0522092022, 0.207347527, -0.0800161883, 0.0155367013, -0.171100616, -0.15568769, 0.0280985534, 0.155661479, -0.0907097906, -0.0465506762, 0.0450913496, -0.167255431, 0.0276872609, -0.0394791812, -0.20365721, -0.135010064, -0.065793246, -0.15259999, -0.24566929, -0.254977822, -0.261519402, -0.123870581, -0.197444856, -0.12559481, 0.179250687, -0.00984245725, -0.0307493377, -0.0284540262, 0.0870079026, -0.101884559, 0.167557895, 0.16733788, 0.0386115685, -0.186165556, -0.0420892499, 0.132793337, -0.0517253689, 0.0506563708, 0.181324065, -0.230184272, 0.172225639, 0.0384657383, 0.201920986, 0.227207035, -0.140594408, 0.0149281584, 0.0272123087, 0.0511507243, 0.157599419, -0.12310376, 0.0275888201, -0.119697392, -0.133497775, 0.177538306, 0.287879407, -0.332083166, 0.174466282, -0.0631491616, -0.0642071292, 0.0698080435, -0.194340572, 0.174546167, 0.112725794, -0.130530342, 0.0916617587, -0.0443805419, -0.242965654, -0.259136677, 0.200497359, -0.16344808, -0.0397210233, 0.0303804427, 0.146784887, 0.15142341, 0.138190344, 0.246435046, 0.077768594, -0.080286853, -0.204465911, -0.0890383646, 0.0499912277, 0.106659219, 0.261487067, 0.16590409, 0.179442301, 0.140036687, 0.0401791185, 0.00325127738, 0.013187293, 0.0925546288, 0.07011462, 0.165935919, -0.256534755, 0.0718082935, 0.0792537257, 0.030161446, 0.242915824, -0.0511688851, -0.0652604699, -0.0842846036, 0.108259201, -0.128864169, -0.00321713765, -0.184777811, 0.0591468774, -0.107330173, -0.0423216075, 0.19637309, -0.107558452, -0.200378031, 0.0274944436, 0.047395166, -0.194123879, 0.188412562, 0.199617177, -0.141710162, 0.221462101, 0.209144309, -0.0284675043, -0.244087934, -0.183096975, -0.0241368171, -0.148103431, 0.177265957, 0.186891973, 0.0422130674, -0.344164699, -0.0773528889, 0.141355872, -0.373026252, 0.0433265753, -0.210413083, -0.148437619, -0.0495266616, -0.17753464, -0.1127683, -0.113730326, -0.156939805, -0.224368513, -0.104205146, -0.0880409703, -0.173214465, 0.0337923206, 0.300643057, 0.00617149146, 0.155847415, 0.126247868, -0.133445188, 0.015533735, -0.183959901, 0.0210792925, -0.192985684, -0.0331071578, 0.135724992, 0.211360231, 0.133701399, 0.0228303764, -0.05452976, 0.110739149, 0.183961943, 0.0661156029, -0.00822394434, -0.11427819, 0.245802104, 0.14801845, -0.0657031313, -0.236966819, -0.207826287, 0.0913634151, 0.0438724905, -0.18313092, 0.00411039777, -0.126928151, -0.211722925, 0.214022741, -0.128302187, 0.0836230144, 0.164736882, -0.112882853, -0.11854811, 0.19892104, -0.207083598, 0.0527174808, -0.0543283299, 0.103308566, -0.142663166, 0.112300202, -0.14731279, 0.0822475776, 0.0341244563, 0.0138530098, 0.073856324, -0.196735963, 0.154973254, 0.233334199, 0.0869767517, 0.116376385, -0.0416299328, 0.0994379148, 0.166396573, 0.16971387, -0.173807308, 0.213895455, -0.0528170429, 0.0617500283, 0.259949446, -0.0118162651, -0.234531507, 0.0625089556, 0.0717810541, -0.13730064, 0.239427283, 0.0305171944, 0.23850891, 0.2220653, 0.25341624, 0.171295524, -0.0135789579, -0.209433094, -0.0696900189, 0.0471944325, -0.138306618, 0.157414973, -0.149076745, -0.149825826, 0.0214383248, -0.118996307, 0.119986966, -0.0147008747, -0.237432435, -0.076058656, -0.0901724845, -0.132154062, 0.0539183468, -0.0170942433, 0.0179768484, 0.22421883, 0.0985278562, 0.228690475, 0.0216967724, -0.131215245, 0.135511026, 0.258222163, -0.0243793726, 0.123374104, 0.129674554, -0.0193014108, -0.143381625, -0.161064699, -0.172403276, -0.158084139, 0.0584857427, 0.0655151159, -0.160059884, -0.204120889, -0.0126833543, -0.0621461421, 0.142932773, -0.0626193658, 0.16576916, -0.15621151, 0.00211782986, 0.103418313, 0.0376950353, 0.0308611691, 0.0366130322, -0.139915824, -0.104231551, -0.207542226, -0.064083159, -0.145862356, 0.146586224, -0.0424620397, 0.186795101, -0.158907622, -0.110902712, 0.142597273, 0.0426524207, -0.011229001, 0.210712969, -0.0741818473, 0.086176455, 0.252430946, -0.123034984, 0.0468166359, -0.134075209, 0.0980751961, -0.0789282247, 0.148234606, 0.105269954, -0.168516472, -0.161657631, 0.0963762105, 0.163820669, 0.135545686, -0.079741396, -0.195735767, -0.077804029, 0.171317056, 0.126934454, -0.0572446063, -0.21873033, 0.21519053, 0.170210302, 0.124228232, -0.073779501, 0.176543459, -0.0158718117, 0.00454410026, -0.118912876, 0.162831694, -0.174594507, 0.0981904119, 0.188442662, 0.0812480599, -0.0692835823, -0.0890745521, 0.0326154418, 0.167388737, -0.03485322, 0.0143670244, 0.0791173428, 0.134169146, 0.0797807947, 0.14800404, -0.141179651, -0.016895188, 0.154919192, 0.00256294012, -0.192573935, 0.118427344, 0.107221924, 0.151232108, 0.210011765, 0.0565974601, 0.00145513611, 0.0219323114, -0.189139843, 0.06658151, 0.21069631, -0.0141648222, 0.0961672589, 0.19676432, 0.11270266, -0.092723079, 0.039994482, -0.0988364965, 0.186328426, 0.0684169978, 0.0352716595, 0.0923228562, -0.247896671, 0.0594582744, 0.215583935, 0.0443359576, 0.106910646, -0.09841194, 0.0154830469, 0.186022297, 0.122082792, 0.109951109, 0.178713337, 0.185618713, -0.00407085847, 0.14384532, 0.237962916, 0.0404084362, -0.162489235, 0.0169203728, 0.0621280223, -0.159193203, 0.120504037, 0.243941158, -0.153041452, -0.133457929, 0.290807456, -0.0554177649, -0.162622347, 0.186095059, 0.0159069337, 0.226315305, 0.192118213, 0.279498637, -0.1455594, -0.360007048, 0.156156048, 0.0351749025, 0.309243917, -0.00659387093, -0.0777715594, 0.212203711, 0.107820228, -0.191825479, -0.215385392, 0.145686373, 0.250261635, 0.132179976, 0.0784063116, 0.141661942, 0.0102276588, -0.28464517, -0.0189468563, -0.153701648, -0.150468856, -0.016683815, 0.133815899, 0.334772259, 0.0575955845, 0.042229306, -0.224532291, -0.0747981966, 0.0232652463, 0.25478974, -0.157321453, 0.133630514, 0.0333518349, -0.266530663, -0.0646840036, -0.172265172, -0.189026609, 0.0687507093, 0.00638828939, 0.319402933, 0.122809738, -0.0131080216, 0.135142997, 0.102929942, -0.202861682, 0.0329007581, 0.00744347926, -0.21400103, -0.316629291, -0.374617159, -0.319015384, 0.384847909, -0.186712921, 0.0658086613, 0.032412149, 0.0714035854, -0.255016744, 0.0262498483, 0.0766730756, 0.138087109, -0.0706778392, 0.0776452422, 0.0143215396, 0.00803621765, 0.152218983, -0.0326965526, -0.233084202, -0.0957412347, -0.182263479, 0.161254615, -0.130365536, 0.0748982504, -0.149099216, -0.215250716, -0.117837511, 0.0308287051, -0.167285755, 0.142437562, -0.0721527189, -0.0916155428, 0.218848243, 0.0761095062, -0.175035179, 0.103456758, 0.20379065, 0.225135043, 0.158203647, -0.142868116, -0.173013821, -0.00321286987, -0.0699528158, 0.107067905, 0.197857693, 0.181346416, -0.133046284, 0.0340469182, -0.0929345265, 0.0420503095, 0.0250554103, 0.184311718, 0.174113616, 0.220722213, 0.00232743588, -0.150735736, 0.0382508636, -0.129761532, -0.130726188, 0.119928777, 0.0578796864, 0.0282058474, 0.0902101099, 0.0399041548, -0.155804977, -0.120978624, 0.249803692, 0.0158650391, 0.0688268542, 0.134503469, -0.288924664, 0.176216707, 0.00563906645, 0.102420114, -0.0788406879, 0.213966206, -0.154680684, 0.0656312183, 0.0721544251, 0.173323125, -0.147119582, 0.0787703097, 0.0888866857, -0.0924119502, -0.0353752673, -0.0151055222, 0.0759745687, 0.280328214, -0.129063725, -0.0747397095, -0.203125596, 0.227080092, -0.206261814, 0.119735092, 0.0916555002, -0.0724879056, -0.155287698, 0.0132731264, 0.212116286, 0.0839198157, 0.114934556, 0.160972327, 0.185490161, 0.182898089, -0.15434128, -0.0223024506, 0.0369399376, -0.242618233, -0.04812406, 0.124690734, 0.0266579203, 0.0357043222, -0.0241595097, -0.170285985, 0.198587388, 0.153542444, -0.0928277895, -0.0493879616, 0.0720407665, -0.0875376537, 0.0800556913, -0.106703565, -0.188763604, 0.1804066, 0.190824226, 0.139410958, 0.134015784, 0.0551224127, -0.0588871315, -0.172435537, 0.120842956, 0.102679841, -0.0483263209, -0.0404443517, -0.0905011818, 0.00734967226, -0.175017715, 0.253821075, 0.107986726, -0.0605778471, -0.127831027, -0.0520662367, -0.15249005, 0.0787140727, 0.177878886, 0.0623937584, -0.0510694347, 0.162456274, 0.0961652696, 0.156488523, -0.0103794681, 0.298527658, 0.117508285, 0.00845222175, 0.00402975967, 0.244920164, -0.262802303, 0.239384681, 0.194349378, -0.0255465209, -0.0071021365, 0.0496552289, 0.189110205, -0.0734819695, -0.0138057666, 0.22511366, -0.024540307, 0.0501983725, -0.130734563, 0.261949658, -0.129572645, 0.0852468386, -0.195301205, -0.128256202, -0.146074802, 0.114428394, -0.109575629, -0.171998858, 0.1805114, -0.0983749181, 0.168353647, 0.00222684909, 0.107877977, -0.133522928, 0.0821961313, 0.055921942, -0.189155638, -0.211974889, 0.035456989, -0.03801715, 0.151340604, 0.0116558271, 0.0453454293, -0.138027087, 0.165734008, 0.0903293639, -0.17851457, -0.181823134, 0.105536416, -0.00437751412, -0.0242398828, -0.197221443, -0.169698417, 0.00265513361, 0.119570628, -0.0556186885, -0.179043248, 0.0923377424, 0.0260195583, 0.142739668, -0.0102109313, -0.0621111393, 0.207488343, 0.0741483122, 0.158786342, -0.101714008, -0.185144261, 0.16310133, 0.0921799093, 0.0151199698, 0.0675591677, 0.0690498203, 0.0627175122, -0.156824663, -0.0990713686, 0.0945287794, -0.0230718404, -0.0956377164, -0.203232855, 0.193041012, -0.171600953, 0.00985047221, -0.0484160632, 0.0128556937, -0.0141810179, 0.199574545, 0.0574304312, -0.0120507926, -0.10293258, 0.171099111, 0.0624095947, 0.127719328, 0.0310608298, -0.127090856, -0.135603577, -0.0402774811, -0.00777311623, -0.0236091018, 0.115270123, -0.0440471768, -0.0969943702, -0.0702738315, 0.00185018778, -0.135444164, 0.138630465, 0.206673846, 0.0269248039, -0.194600731, -0.108348511, 0.100241527, 0.204216614, 0.0310706943, 0.0207177736, 0.0246665124, -0.0369903184, 0.189978585, 0.18308571, 0.0601348951, 0.165929869, -0.0339035504, -0.0099209277, 0.190639094, -0.13286522, -0.00495153386, -0.0395436101, -0.138987705, 0.176830545, 0.00814937707, 0.252283871, 0.218431175, -0.0865562707, 0.0898508579, -0.0586666316, 0.155118331, 0.0155698694, 0.178617969, 0.0938429683, 0.0607920587, -0.209286168, -0.142663464, -0.104432322, -0.207258865, 0.128569424, -0.0403374508, 0.0755493268, -0.123791821, 0.166542724, 0.103759401, -0.260609299, 0.0588776469, 0.163806662, 0.00261614448, -0.00516588986, 0.0550476126, -0.34296912, -0.12214759, 0.163169816, 0.0452847183, 0.178035349, -0.0292446893, 0.00157334586, -0.143873423, 0.129343823, 0.214960068, -0.062136814, -0.0185418073, 0.185974956, 0.050098747, 0.20793201, 0.228919804, -0.174892411, 0.0396745056, -0.129953608, 0.206800371, -0.000112072892, -0.138918951, 0.0954689011, 0.255405635, -0.118499793, -0.175630018, 0.123674139, 0.0513064191, 0.236296624, 0.0593134351, 0.0739371106, -0.0461705178, -0.106488623, 0.128243804, -0.229913831, 0.103818499, -0.208989188, 0.0269889422, -0.0170714278, 0.172011673, -0.00835058093, 0.083449766, -0.153386265, -0.206975192, -0.0904331207, -0.100907929, 0.0201056469, 0.0092816418, 0.138591155, 0.123229094, -0.204459578, 0.125524312, -0.198420554, 0.136316523, 0.0642325506, -0.111182407, -0.292572588, -0.0476938225, 0.25313285, 0.0092351269, -0.0328827761, -0.112535074, -0.0818377212, 0.143190131, 0.162059993, 0.0104096029, -0.0401865542, 0.072995171, 0.204331324, 0.0964775011, 0.0549218319, -0.26574558, -0.149334505, -0.219716296, 0.0813605562, -0.102174677, 0.165653527, -0.23237288, 0.0617746599, 0.219712645, -0.245772511, 0.0843116418, -0.0313958414, -0.0511075445, -0.202375591, -0.0243414436, 0.0134311467, -0.184688628, 0.0857788771, -0.0375306755, -0.212528273, 0.0812165588, -0.14801389, 0.103163257, 0.124996766, -0.112198733, -0.214695185, 0.196181044, 0.0699417144, -0.214553803, -0.158492222, -0.173867494, -0.040612489, -0.0375947803, 0.060765788, -0.0616895109, -0.0461635143, 0.215136424, -0.158336386, 0.0892048329, 0.0994321257, 0.113832906, 0.20994629, 0.0749067515, 0.0561294109, -0.0114479363, -0.117390744, -0.0267652422, -0.152938411, 0.13877742, 0.104254767, -0.169561014, 0.180426642, 0.111701086, -0.00645264983, 0.125381544, -0.147052184, 0.153655097, -0.0217939615, -0.0914004594, -0.178690523, 0.178770587, -0.0424079597, 0.024468869, 0.0716981441, -0.119676486, -0.0311208218, -0.0731271207, -0.103556246, 0.0954664797, 0.0873899013, -0.0905441493, -0.144235373, -0.0789919347, -0.10910587, -0.0982930511, -0.0370353907, 0.189428493, 0.00647680461, -0.0638864785, 0.212589487, -0.161814377, 0.0216575265, -0.0850141943, 0.194710687, -0.178992704, 0.125666514, -0.192258149, -0.193372041, 0.20426394, 0.118718341, 0.100960627, 0.0680707842, 0.0463458747, 0.165338323, -0.0671609789, 0.168787971, -0.0070540607, -0.202503204, -0.0853080601, 0.211600348, -0.122439608, -0.147218913, 0.199023679, 0.120119318, -0.0956019461, -0.122479819, 0.0545401126, 0.214297399, 0.0260116011, 0.117337689, -0.182416037, -0.0304358751, -0.194916844, -0.0680961162, 0.0540857166, 0.176674083, -0.0712954253, -0.00287421048, 0.0383953899, 0.0185558945, 0.112168685, -0.180515826, -0.112304345, -0.0206410438, 0.0596600622, 0.0638618618, -0.148700684, -0.181752264, -0.206867248, 0.142111555, -0.0103422552, 0.16394259, 0.199925497, 0.208245948, -0.125069648, 0.0724749714, 0.132800862, 0.131532744, 0.122560248, 0.0359630138, 0.0514701158, -0.00991392136, 0.16258727, -0.102539249, 0.131538868, 0.000688975444, 0.210872754, -0.0939219445, -0.155480877, -0.0926667899, 0.150634632, -0.125974014, -0.0297515579, 0.0463272557, 0.0345584452, -0.159411788, -0.00879441015, 0.0906654373, -0.222819507, 0.300452858, 0.24445796, -0.220637038, -0.073617816, 0.0579014607, 0.160616696, -0.179756835, -0.0254850835, -0.136787683, 0.0766259208, 0.120203525, 0.149309546, 0.168427154, -0.0670610815, -0.104210295, -0.112162739, -0.101194017, 0.124157779, 0.121481434, 0.176228672, 0.172684014, -0.166508585, 0.0264002513, 0.0834020749, -0.182705998, 0.112678163, -0.0141648045, 0.00864631962, -0.135217071, 0.139958009, -0.111488022, -0.0717050955, -0.21887809, -0.0830352902, 0.106444001, 0.194088787, 0.0767873973, -0.150106505, -0.0719411075, 0.0724190921, 0.292881131, -0.0399664752, 0.243576974, 0.117913261, 0.246021658, 0.0811332464, -0.0399341844, -0.0816165209, 0.171891883, 0.082011655, 0.0575862974, -0.109388068, -0.163562402, 0.170695201, -0.162173331, -0.134208307, 0.158017829, 0.163954869, -0.198981807, 0.133076355, 0.174984023, 0.0209734291, -0.135800138, 0.167734668, 0.190667316, 0.203086928, 0.146870956, 0.0645530969, 0.113435879, -0.187958598, 0.147743359, 0.0670311004, -0.187562466, -0.0608942211, -0.0351307988, -0.058291018, -0.129617661, -0.0873317271, 0.0594988018, -0.211554736, -0.0564201325, -0.128696471, -0.0596370399, -0.181903094, -0.153074175, 0.0677614063, -0.08287628, 0.113757566, -0.153864205, -0.00586368144, -0.216033623, 0.0404614061, -0.214554414, 0.100273564, 0.139342979, 0.0685483068, 0.129975602, -0.173656166, -0.0469692796, 0.135614976, 0.188055262, 0.127508983, 0.0973801762, 0.116156682, 0.0537556559, -0.0190902501, 0.0643442422, -0.176481023, -0.0268422067, 0.170466408, -0.0452373028, 0.0346771628, -0.0764650702, -0.161790356, -0.169284806, -0.160289347, -0.0043374598, 0.0272316784, -0.0586752929, 0.0605526119, -0.175261557, 0.159667954, -0.139275417, 0.187538177, 0.0448392779, 0.0851275474, -0.0254395697, -0.168208286, 0.205435231, 0.0792442113, -0.167214826, -0.162651837, 0.0390271097, -0.0277169496, -0.0349142514, 0.122520849, -0.129117578, 0.116114929, -0.0394956619, -0.131158963, 0.0104077011, -0.183592737, -0.0942491591, 0.0787120685, 0.0059645921, 0.083924517, -0.00701065361, -0.118871383, 0.140056029, 0.211868882, 0.0615758449, 0.00838501751, -0.000891566277, 0.0594077855, 0.146011487, -0.0805511698, -0.193798214, -0.186887994, -0.089735806, -0.180153847, -0.0625011772, -0.123947091, 0.194204822, 0.00806425512, -0.116187446, 0.0269125104, -0.0904725119, 0.011333555, -0.0565276444, -0.166684598, -0.17863436, -0.184847683, 0.206926495, 0.199473783, 0.028638497, 0.0610053949, -0.209566385, -0.149408638, 0.0373195261, 0.06447687, -0.126612946, 0.28914547, -0.0355662853, 0.0583788455, -0.2373074, 0.221651822, 0.175030649, -0.0361175053, 0.154063821, 0.242598936, 0.178581849, 0.13535817, 0.0564856976, -0.0409523547, 0.106473468, -0.0620523989, 0.146483317, 0.0771263912, -0.165507808, -0.0569170639, 0.214328185, -0.0147469528, 0.146464691, -0.0852415189, -0.0795736313, 0.0171650928, 0.262713403, -0.0182778351, -0.125869542, 0.218170211, 0.08039435, 0.166997373, -0.0870893747, -0.104434751, 0.135473803, 0.0149303246, -0.0789194182, 0.279207557, -0.232716322, 0.0479517728, 0.111858115, -0.0409652069, 0.120025121, 0.0328806192, -0.234696463, 0.109781213, 0.242693588, 0.263724536, -0.209186554, -0.0229675435, -0.177582771, -0.134655267, 0.301631212, 0.173010796, 0.277582735, 0.0801606327, 0.115403861, 0.258175075, -0.203490555, -0.169273093, 0.197581336, 0.233946189, 0.188818827, -0.110022955, -0.0721238554, -0.127027333, -0.0361180678, -0.182209134, -0.0469776765, 0.0636565313, -0.125594214, 0.112164833, -0.153257549, -0.0699059218, 0.0906096771, -0.156303734, 0.163650781, -0.120070562, -0.187784672, -0.110630184, -0.0369865112, -0.221759483, 0.265062481, -0.0200742166, -0.0210180636, -0.0318562686, 0.289968342, 0.209271714, -0.163250521, -0.033234816, -0.158912554, -0.15139316, -0.161861673, -0.182225049, 0.0245842095, 0.0447209552, -0.133103281, 0.0522985011, -0.140202329, -0.0881955624, 0.0748139471, 0.14398168, 0.229476035, -0.100793242, -0.0547418669, 0.254428893, -0.0232664496, -0.0325468257, -0.118670925, 0.167250693, -0.220140129, -0.0891620591, -0.0795891732, 0.125988051, 0.360238761, -0.187357172, 0.164008111, -0.184598282, -0.250819564, -0.0614155643, -0.213410959, 0.0295955334, -0.188740283, 0.165933087, 0.14575623, -0.169412017, 0.0403924398, 0.0863903165, 0.125428617, -0.122938238, 0.203624532, 0.0290758889, -0.194397897, -0.0813511461, 0.136541203, -0.168952912, -0.118765511, 0.07683599, -0.129231229, -0.0414971858, -0.0406129733, 0.101526216, -0.0764528364, 0.131897673, 0.0560044497, -0.0730934143, 0.0276858192, 0.173554912, 0.00495803775, -0.0322014466, -0.0102797113, 0.213982448, -0.0208447874, -0.107821919, -0.0264427457, 0.0145503255, 0.019508658, 0.0594968982, -0.0592152774, 0.121941999, 0.122733139, -0.140440956, -0.176466525, -0.0972242281, 0.0811412483, -0.212435484, -0.107308395, -0.0842584148, 0.0197450221, 0.215222329, 0.17154865, -0.0421809405, -0.0426143073, 0.156440645, -0.123030953, -0.0165297743, 0.086967513, 0.130930915, 0.192302629, 0.108801588, 0.189616874, 0.134053215, -0.100600176, -0.105523147, 0.0837425441, 0.176915631, -0.0862870663, -0.128423661, -0.185953289, 0.162213311, 0.238823578, -0.0322427824, -0.172987208, 0.0383077003, -0.168837801, -0.0999560133, -0.140007496, -0.13302283, 0.0654487237, -0.054558441, 0.00409579836, -0.0385583751, 0.0616787598, 0.0229705647, 0.174310103, 0.220073834, -0.228525922, 0.20903562, -0.12730284, 0.266811848, -0.0645477623, 0.12383756, -0.11437133, -0.110793918, -0.0366560929, -0.113584034, 0.0970615298, -0.0828079358, 0.186074406, 0.16188024, -0.0919989794, -0.0214854963, 0.209291995, 0.132674858, -0.158335567, 0.129601404, -0.043703422, -0.0580179356, -0.122194469, 0.0626526251, 0.0995965749, 0.125470623, -0.173571438, -7.04564809e-05, 0.0105728703, -0.142664522, -0.0462249145, 0.0775359049, -0.0809029341, -0.13692227, -0.0882295668, 0.0266289487, 0.0734391138, 0.0406049676, 0.192088261, -0.0451808535, -0.0661438555, 0.120225728, 0.151128128, -0.10713999, -0.0322566256, -0.134458154, 0.0705581233, -0.200856641, -0.113959946, 0.161113799, -0.181794733, 0.15956901, 0.160805613, -0.186158001, -0.0237688925, 0.127835721, -0.0186184216, 0.101857841, 0.197322085, 0.125265792, -0.01271844, -0.171266645, 0.0350334905, -0.108482718, -0.214593604, 0.172298625, -0.182126477, 0.161291301, 0.146099284, 0.103996262, 0.0945375413, -0.212611616, -0.150450736, 0.155232683, -0.0679181367, -0.155561522, -0.0921959952, 0.0946691111, -0.127165928, -0.122972131, -0.186263174, -0.139322162, 0.242685571, 0.0045821243, 0.011791165, -0.0878160745, -0.159043938, 0.0593511797, -0.167231545, 0.23195985, -2.63589227e-05, -0.150773689, 0.0332254022, -0.115814731, -0.191897079, 0.104204178, -0.0777447969, 0.17065756, -0.217323199, 0.114431463, 0.069135122, -0.0210048091, 0.00420680922, -0.0845233724, 0.0959770456, 0.0833298042, 0.0301761869, 0.0593393333, -0.158845872, 0.0165265705, 0.0481217168, -0.00209004036, 0.138400525, 0.1577003, -0.206650645, -0.140175536, 0.139429837, 0.0434673727, -0.00637131557, -0.150466055, 0.0634823367, -0.122112915, -0.115015678, 0.0883953124, 0.213094011, -0.128786102, 0.10067419, 0.269909352, -0.0107553555, -0.135354757, -0.217162892, 0.0356924273, -0.0991727114, 0.132911071, -0.0588454865, 0.243446231, -0.254837215, -0.0441369563, 0.0588260442, 0.174045861, 0.0421890616, -0.0813888386, 0.280730367, 0.255607665, 0.208496362, 0.256909579, 0.0790268704, -0.118365906, -0.21108976, -0.135365918, -0.191761851, 0.147386804, -0.238638878, 0.0442762636, -0.106006496, 0.0480982736, -0.262756944, -0.083258003, -0.210455641, 0.221321031, 0.214391738, 0.140733302, 0.168415472, 0.177380338, -0.0998223275, 0.0802876726, 0.024429664, 0.23944816, -0.0581545308, 0.213931069, 0.196635291, -0.0161537938, -0.0103867967, -0.126716629, -0.083251968, -0.0781524554, -0.0834515467, 0.0193810612, -0.186825454, -0.128707543, 0.204980001, -0.00399512053, -0.101887874, 0.0210454538, -0.0412895195, -0.0971676558, -0.048628062, -0.20430325, -0.197556436, -0.190492779, 0.0837618262, 0.125030011, -0.0541782528, 0.146718219, -0.150529712, 0.113789588, 0.159004748, -0.00630572857, -0.206578702, 0.167073652, -0.0800563917, -0.0184968971, -0.132193252, 0.15642193, -0.146631718, -0.0564464815, 0.0205936134, 0.215904519, -0.170073912, 0.0835290179, 0.00320865051, 0.0229984596, -0.114689462, 0.171532705, -0.0459926128, 0.057841301, -0.0879666209, -0.0287654698, -0.144966319, 0.105421446, -0.0273225829, 0.0585521348, -0.101430416, 0.131310791, -0.0334190056, 0.184861079, 0.0362242311, 0.205380991, 0.0049544517, -0.0775810778, -0.21244362, 0.0842021108, 0.0351231582, -0.181801394, -0.0861293525, 0.0863052607, -0.0654114634, 0.0168641414, -0.0446151756, 0.247980848, -0.122818522, 0.182896554, 0.0511074699, 0.0474656112, -0.133897036, -0.157300696, 0.131089389, 0.00570026645, 0.156846672, 0.0670417845, -0.074737817, 0.179072648, 0.139402583, 0.209800005, 0.0514971539, -0.157501861, -0.137726873, 0.0395912975, 0.0381566659, -0.0413452275, 0.046529077, 0.195759162, -0.0611983314, 0.0869912729, 0.16404058, 0.197312593, -0.185774952, 0.172979549, 0.269182414, 0.0887734294, 0.205442265, 0.01246008, -0.211092308, 0.227946341, -0.0107464157, 0.245333567, -0.048793897, -0.0402365625, 0.0947469473, 0.0884542614, -0.0422119237, 0.165364295, 0.0160138234, -0.0176507104, -0.178265303, 0.0195886772, -0.0455894843, -0.0993135348, 0.0292526782, -0.0872291252, -0.194193006, -0.204600781, 0.144727439, -0.265376478, 0.262558103, 0.0440654457, 0.00297656655, 0.124401599, 0.256192356, 0.140282795, 0.181511864, 0.127582431, -0.0810992941, 0.00457523856, 0.194761962, -0.0414959528, 0.0110664666, -0.0478526093, 0.218107626, -0.097522147, 0.0221662484, 0.0307420697, 0.00897521432, 0.0723016262, 0.156312093, 0.0830891505, -0.102879122, -0.220429748, 0.111000456, 0.0493231416, -0.167957768, -0.200361371, -0.220628932, 0.0213064477, -0.13790077, 0.16264008, 0.0366902873, 0.0662807301, 0.0843776241, -0.00975239743, -0.187409461, -0.00850835908, 0.214093223, -0.0262640547, -0.0037057586, 0.261299968, -0.0119852293, 0.0840612352, -0.140529484, 0.086045213, -0.178673238, -0.101949222, -0.0606811792, 0.2623505, -0.159947217, -0.152141213, -0.0400353037, 0.0315761305, 0.1173632, 0.117560208, -0.0394015647, 0.194363236, 0.0334627554, 0.122356705, 0.0350546427, 0.0978516936, -0.236527696, 0.205010638, 0.248273745, -0.0951982066, 0.0346223675, 0.07659439, 0.0673788562, -0.0866984576, 0.0852876976, -0.069079563, 0.019739734, -0.0612785369, -0.103156194, -0.131891444, 0.194864705, -0.194438815, -0.132523477, -0.202051356, 0.0380129889, 0.137692869, -0.100640491, -0.0755962133, -0.12461704, 0.0515572987, 0.132496744, -0.0181591716, -0.146472231, -0.118328683, -0.168681785, 0.0452108234, -0.196983844, -0.133911699, -0.107775599, 0.0720314309, 0.139389187, -0.127528727, -0.114843562, 0.140681937, -0.208352178, 0.0613223463, -0.0877515376, 0.0889104754, -0.122407876, 0.0725748539, 0.0339392349, 0.0478396267, -0.198128894, 0.0607758276, -0.0642398596, 0.119521871, 0.206692919, -0.0587804914, 0.205643147, 0.108449683, -0.100034304, -0.158070832, 0.116327606, 0.0159044266, -0.102844685, -0.0278574713, 0.160228476, -0.175503105, 0.194432482, -0.192663267, -0.0688776821, 0.20138903, 0.11521215, 0.0320747495, 0.0258750096, 0.182264447, 0.0569877252, -0.0823236406, -0.0462619513, 0.106567733, -0.0499362051, 0.0560031161, -0.00147831102, 0.215228215, 0.102208264, 0.22965087, -0.0239753295, 0.095687367, -0.0616672896, 0.0587593913, 0.151922241, 0.0286311377, 0.0363215096, 0.115954399, -0.0627551451, -0.0331935957, -0.0891616046, 0.0451479107, 0.0505939499, -0.201272562, -0.0867501497, 0.152432233, -0.234590366, 0.142962754, -0.0309544504, 0.0265288632, -0.107768282, 0.0372548141, -0.185375005, 0.0994121656, 0.146933943, -0.0775678679, 0.136601061, 0.116011761, 0.162975177, -0.133521244, 0.0610307641, -0.172060072, -0.175027579, -0.0902606323, -0.119711854, 0.00174348196, -0.080424875, -0.0717453212, 0.0530059896, 0.142690092, -0.2024865, 0.0607569851, 0.0632190183, -0.0805430338, 0.0256457161, 0.202368066, -0.182796001, -0.22332494, -0.173913211, -0.0483726896, 0.130500004, 0.14105849, -0.0087418789, 0.0575943477, -0.0352024697, -0.0449910536, 0.0370082781, 0.0126874121, -0.143768162, 0.0430835038, 0.0192103907, 0.214269981, 0.121653453, -0.171620205, -0.115121514, 0.0637972057, -0.150997698, 0.138255328, 0.0768500865, 0.0764330328, 0.205035627, -0.203529269, 0.144700333, -0.134389654, 0.208693668, 0.0657688901, -0.068395406, -0.0664896816, -0.113522142, -0.0315324329, -0.0550373867, -0.0346781798, -0.145656422, 0.0172823854, -0.0111174863, -0.157122552, -0.190427795, -0.0916103199, -0.00143183256, 0.0899138302, 0.136021599, -0.198203564, 0.174707979, -0.0790932477, 0.134556785, 0.0119398087, -0.0647746325, -0.0214638021, -0.0843484104, -0.112631276, -0.0474717468, 0.0715068504, -0.0579168312, -0.0775391087, -0.0880511031, 0.0911753923, 0.0051047653, -0.150063142, -0.0598085932, 0.0396242812, -0.0492532253, -0.091608271, 0.150526419, -0.0564503483, 0.0292801782, -0.0795698985, 0.0905861259, 0.154940531, -0.0895984471, -0.158532158, -0.0644570738, -0.0941605195, 0.0961572528, 0.27700609, 0.0923415422, 0.157652989, 0.0674565509, -0.0285261758, 0.0780545026, -0.150813326, -0.078189984, 0.0764895827, 0.140417024, 0.176455826, -0.0467667431, -0.0611154847, -0.135509744, 0.0651874691, 0.00128756708, -0.13219206, 0.0725255162, 0.0488932282, -0.211957008, -0.241675302, -0.0976792723, 0.079120189, -0.0794882551, 0.0674599707, 0.306206286, 0.167326748, -0.0135372728, 0.256001234, -0.222973049, -0.0457991101, 0.0760016367, 0.174197108, -0.0268575419, 0.0531892926, -0.0637947321, 0.199966535, 0.0592058152, -0.166631758, -0.0820748508, 0.044286795, -0.0869615451, -0.0670766756, -0.0154077159, 0.168325067, 0.0498711281, -0.0202831142, 0.178866312, -0.253515154, 0.122428641, -0.0470641106, -0.180592746, -0.193016753, 0.198658079, -0.0529388189, 0.108853698, 0.0329008251, -0.172148854, 0.155390486, 0.223928601, -0.105937399, -0.109959118, 0.256064564, -0.107306272, -0.119646482, 0.0797421783, 0.0929884836, 0.0979342908, 0.133596629, -0.0257349536, -0.198378071, -0.109671965, -0.140990347, 0.0564259849, -0.00328065758, 0.0223205835, -0.111956462, 0.100838266, -0.118380174, -0.106406175, 0.13367115, 0.140827075, 0.149365082, -0.034094438, -0.0994511619, -0.202903464, -0.102243468, 0.216089889, -0.167881742, -0.185640097, -0.163032368, 0.0955848545, 0.196899727, 0.198177576, 0.189767465, -0.125597715, -0.0851550102, -0.012896874, -0.0585481524, -0.12292812, 0.161586598, -0.10934332, 0.0761391968, 0.00712056924, 0.0470088422, -0.0579094887, -0.00209463271, 0.0494624302, -0.00159580936, 0.126086533, -0.029434476, -0.0511376858, 0.0322339237, 0.0604848899, 0.217367649, -0.157550901, -0.1742405, 0.00597815914, -0.181396201, -0.0200733002, 0.0123654017, 0.212862641, -0.0284591522, -0.0449727364, 0.168478563, -0.0509453565, 0.112934813, -0.0566788465, 0.176471725, 0.0360399634, -0.0752981752, -0.146713302, 0.115039334, -0.128386751, -0.0662233233, -0.046212554, -0.0662843436, -0.126971036, 0.116823152, 0.191384241, -0.0919323936, -0.0727686882, -0.173104316, -0.0298395753, -0.131576031, 0.145610556, -0.016514197, 0.089529559, -0.1694635, 0.0887180716, 0.0909219533, 0.206983224, -0.128153592, -0.175801769, 0.156361684, -0.141585872, -0.0933236778, -0.0274668038, 0.200519279, 0.16725488, 0.0719681829, -0.0101237446, -0.189104065, 0.203866377, -0.140116215, 0.168043867, -0.0233105272, -0.202382937, 0.13448818, -0.0404603183, 0.0488183945, -0.0125396252, 0.0655785948, -0.0455810428, -0.131461859, 0.0987256318, -0.0785749108, 0.0762815624, 0.0706483275, -0.182909623, 0.204016224, -0.0563442409, -0.161886901, -0.204789057, -0.0380925536, 0.149280533, 0.186354056, -0.142447859, -0.190923437, 0.0317074656, -0.195126057, 0.0115836412, -0.0849219933, -0.00952991843, 0.0764236376, 0.0596605688, 0.120444655, 0.184710845, 0.0115267038, 0.127696022, -0.146930456, 0.169530034, 0.0189637188, -0.021946907, -0.0109692765, 0.0416838974, -0.00754594803, 0.0580874756, 0.0444080979, 0.184013709, 0.104757175, -0.0313890278, -0.100590184, 0.128223568, -0.20617266, -0.132255659, -0.0874492675, -0.143805087, -0.0500562638, -0.205596805, 0.148389444, 0.00172358123, -0.106911823, 0.0452977568, -0.21107322, 0.0668992624, 0.122114658, 0.0477002077, 0.120604172, -0.188552618, -0.138453364, -0.0456057191, 0.115633465, 0.165090904, 0.0320103727, 0.0575927421, 0.177304104, 0.0367988423, -0.212701097, 0.195212469, -0.194699734, 0.0594319105, 0.0195149295, -0.210422724, 0.18505533, 0.156053185, -0.0448524803, 0.123860724, 0.0762408525, -0.191941276, 0.113714948, 0.0830711722, -0.162165016, -0.0373560488, -0.118707739, -0.10479752, -0.182017535, -0.151235938, 0.0206096731, 0.145007297, -0.0153894899, 0.218414783, -0.000869259238, 0.0154756503, -0.200680226, 0.170030713, 0.0636367649, -0.172657162, 0.0794806182, 0.150627524, -0.102580756, -0.0683144256, -0.0945177898, 0.102912441, 0.169210717, -0.120361015, 0.194299057, -0.188841209, 0.146587253, -0.188844159, -0.0558344238, 0.0359239876, 0.053900253, 0.0142748058, -0.0113670798, -0.111485705, 0.0116025666, -0.215477005, -0.0928430185, 0.115675338, -0.102832057, 0.168732792, -0.126997501, -0.221014336, 0.182971597, -0.152135015, -0.0638246462, 0.180992663, -0.0825914219, -0.200327739, 0.186104283, -0.0761064738, 0.0455469042, 0.175332025, -0.0451734737, -0.172262177, 0.0572228953, -0.168096662, 0.204400107, 0.00175916846, -0.05636115, -0.163206309, 0.0695815533, 0.0637750551, 0.179285645, 0.018083917, -0.0526664667, 0.0717682764, -0.16865924, -0.150882706, -0.0112172551, -0.11952614, 0.0920963809, -0.115396291, -0.150909141, -0.179976657, -0.0421908833, -0.163812667, 0.122877382, -0.0942356437, 0.0453507863, -0.11259599, -0.0999261439, -0.100916177, -0.182669953, 0.154555917, -0.184113041, 0.0896566585, 0.145971134, 0.197596744, -0.0454761721, -0.150642499, 0.159919247, -0.143244132, 0.0210799035, -0.0441629775, -0.0810907111, -0.163442492, 0.045595862, 0.16091612, 0.106087513, 0.0664898232, -0.135403961, -0.0642762035, -0.174812168, -0.0309586972, -0.0548433885, -0.207458809, 0.172602981, 0.0843047872, 0.00955646299, 0.190302178, -0.0120949578, -0.152737558, 0.231507719, -0.0443149954, 0.0997370183, 0.133509561, -0.15396592, -0.129581988, -0.182943463, -0.169034809, 0.0301441699, 0.0955079123, -0.255378693, 0.0398402438, -0.0638692528, 0.154308721, 0.0580761209, -0.0793571323, -0.0826579779, 0.0314475968, 0.219111726, 0.0478798449, 0.0276127569, -0.00546862464, 0.0695564821, -0.131611675, 0.202782288, 0.183789968, -0.0195452888, -0.13255091, -0.0230764579, 0.111142918, -0.0910572112, 0.056702368, 0.14888303, -0.0929223374, -0.178360641, 0.164307311, -0.0853743032, -0.0649680644, 0.0779206306, -0.119389273, 0.230036467, -0.0436925627, 0.137377337, 0.0679846555, 0.0158325471, -0.0744110644, -0.222410843, -0.168998629, 0.0108635696, 0.183892742, 0.160881788, -0.0410534963, 0.05518483, -0.0880163535, -0.0370547585, -0.00287609058, -0.0478597283, -0.199008241, 0.146402642, 0.171959668, 0.290840656, -0.112652093, 0.105188161, -0.0585999079, -0.0022179212, -0.270577133, -0.0842458159, 0.184451506, -0.133775994, 0.244962484, -0.0110368654, -0.202473283, 0.0172045603, 0.145742238, 0.0488118939, -0.0988596231, 0.151816502, 0.0309539363, -0.0803498104, 0.237187728, 0.137721777, 0.0540012866, -0.00746989995, 0.0480698049, 0.150505424, 0.183417454, 0.0880424529, -0.0611262359, 0.0990205705, 0.155396596, 0.0898856223, -0.0296041518, -0.034501303, -0.0609594285, -0.104777358, -0.0443655364, -0.159524351, -0.0758568123, -0.149849355, -0.107333899, 0.0991479903, -0.122835763, -0.109809339, -0.114645869, 0.194594607, 0.0984508544, 0.23515442, -0.000617691898, -0.128364742, 0.199048966, -0.0401824042, -0.0760140866, -0.11002256, 0.0939248428, -0.05619229, 0.122873552, 0.268885493, 0.103352867, -0.105801336, 0.0070370757, 0.106131047, -0.0532236435, 0.0677729547, -0.123542935, 0.222401768, 0.124410555, 0.181627676, -0.0229594037, -0.138093278, 0.107260153, 0.0116578275, -0.0297462214, 0.1843528, 0.051715672, 0.109194115, -0.0787402317, -0.00220843637, -0.0251405481, -0.121136881, -0.0643095151, 0.203086615, -0.0400864892, 0.0907601193, -0.144587412, -0.0898020267, -0.098853603, -0.0770658627, -0.287551373, -0.0851627141, 0.0827269629, -0.0861964077, 0.0113888374, -0.0776093453, 0.0809763595, 0.0635781661, 0.00109870185, 0.216651306, 0.0141436849, -0.12719737, 0.0942884311, 0.303492576, 0.0959326848, 0.17719087, -0.0954696015, 0.323434025, -0.166302964, -0.0378812701, 0.119964503, 0.222246632, 0.0803848058, 0.0778280646, 0.274888039, -0.1463819, 0.16310896, -0.139771625, -0.180156469, 0.164859727, 0.305645019, 0.25364998, -0.0705485269, 0.135831848, -0.0893951431, 0.28743431, 0.070728071, 0.0838205442, -0.0445251912, -0.0326616764, -0.120599262, 0.139440745, -0.270022005, -0.108915411, -0.0532744862, -0.245501712, -0.0115316864, -0.127213374, 0.149182394, 0.173800245, 0.0761279762, 0.238401845, -0.062345773, 0.0435865968, 0.0119816968, -0.113206729, 0.142904684, 0.0389598235, 0.236816138, -0.058863014, -0.140110746, 0.274992466, -0.14359425, 0.10345877, -0.0460031852, -0.167516112, -0.00952434354, 0.247703657, -0.0753713027, 0.121685714, 0.0823878422, 0.23488979, -0.0619931184, -0.0766328648, -0.0780418068, -0.0143457921, -0.133595392, 0.280221343, -0.123221971, 0.0499226376, -0.0771679506, -0.0386132747, 0.050129544, -0.0213634074, 0.0406502597, 0.29187867, 0.00179839157, -0.128595933, 0.0654454753, 0.0833715722, -0.0237372257, -0.160019487, -0.0706409961, 0.13007459, 0.193477109, 0.12929526, 0.194544196, -0.0337707773, 0.153220907, 0.208017707, -0.112889752, -0.0212976448, -0.110117443, -0.0935627148, 0.201002955, -0.0485042818, 0.135973632, 0.127661034, 0.11343646, -0.1885878, -0.0211448614, -0.126879215, -0.183075756, -0.0898045972, 0.000568327669, 0.00911092758, 0.0558643304, -0.18213293, 0.0719175339, 0.152180195, -0.0481474549, 0.258260578, 0.199615657, 0.148173228, 0.0394268632, 0.10337054, 0.106657632, 0.193686217, -0.113603137, -0.137724444, 0.0699722022, 0.063817814, -0.0267793834, 0.0403312594, 0.0746018738, -0.0369499028, 0.111911014, -0.209794521, 0.124978349, -0.0450591743, 0.114969119, -0.207217485, 0.0647557825, 0.15988557, -0.0394030064, -0.00352300704, 0.07973288, -0.183837622, 0.143634632, 0.0214877576, -0.0452758223, 0.207906798, 0.0875673741, -0.133096695, -0.0591884553, -0.171955109, 0.0771896988, 0.0395951718, -0.0173865706, -0.100543596, 0.202937528, 0.206836805, -0.154319584, 0.027785033, -0.0755964369, 0.0502325445, -0.0981198698, -0.204409614, -0.200881124, -0.0966312289, 0.1947162, -0.205129281, -0.0549425334, -0.13413088, -0.00894080102, -0.132092237, -0.01263915, 0.102246657, 0.183655664, 0.0780696124, 0.147488251, 0.0796844512, -0.206366494, 0.105821297, -0.0866758525, 0.117468521, 0.0730968863, -0.0894768089, -0.197888821, 0.123780325, 0.0636071116, 0.182967439, -0.048382435, 0.309802204, -0.250160158, -0.167235941, -0.203475639, 0.0432632677, 0.175398722, -0.0192775838, 0.100834183, -0.152954876, 0.0144183151, 0.232581377, -0.321812779, 0.167421177, -0.191333041, -0.117632791, -0.214048147, 0.0570586398, -0.0707548633, -0.0965818316, 0.0956328809, -0.211586624, 0.159526497, -0.122753829, 0.0936640054, 0.038983807, -0.0090486221, 0.134821489, 0.167622879, 0.156822473, 0.0900678411, 0.153534383, -0.226792514, 0.0524546355, -0.174388677, -0.115811922, 0.00570448162, 0.27308467, -0.106389359, -0.136367708, -0.222481415, 0.0649660677, 0.231387734, 0.199437037, -0.0451859161, 0.00607657246, 0.122315645, -0.0604027137, 0.126780376, 0.144564077, 0.0225306693, 0.0650955886, 0.0242205709, -0.118545949, 0.268948376, -0.0256855562, 0.0343104936, -0.069202207, -0.0779325366, -0.102411069, 0.179498464, -0.101506397, 0.0488925502, -0.0689219609, -0.0659783483, -0.136400327, 0.133670032, 0.243812606, -0.00633601891, -0.148582682, -0.00797831547, -0.126626313, -0.0936052874, -0.197196543, 0.182358727, 0.116384923, 0.0608248077, -0.114480652, 0.0227467716, -0.0658283457, 0.155729368, 0.239702567, 0.197265238, -0.109269656, 0.048140429, -0.113062605, -0.164667413, 0.109318092, 0.117424659, 0.226807907, 0.242188722, 0.244667873, 0.0913275629, -0.0497324169, 0.133244559, 0.139072567, -0.0962307155, 0.156236574, 0.0416714326, 0.0171999503, -0.115829073, 0.193360731, -0.0875519365, 0.0553654693, 0.15870443, 0.112140588, 0.0085960133, 0.115142487, 0.0321300998, 0.0831481293, 0.0826298743, 0.16946727, 0.1216354, 0.0426968448, 0.0600113608, 0.00731581124, -0.0923310071, -0.0970181897, -0.110141873, -0.0211779475, 0.180789977, 0.214999735, 0.143563792, -0.0888314769, -0.0837424845, 0.19645004, -0.0607952587, 0.0226881709, -0.334903687, -0.0999383703, 0.218144059, 0.213849559, 0.163884476, 0.0333319828, -0.0647564679, 0.138918817, -0.190249652, -0.186543033, 0.214060068, -0.139762402, 0.118343443, 0.200249881, 0.195759326, 0.0673449859, 0.0379764214, 0.226978466, -0.205298588, -0.20902957, 0.153362259, 0.01173349, 0.078916654, -0.100195095, 0.151100561, -0.0188093036, -0.0797100887, -0.233888417, 0.117763057, -0.0822941959, 0.0278804805, 0.143493846, 0.160960034, -0.0659005791, -0.108755261, 0.187783971, 0.0706701577, -0.188152313, 0.0074400031, 0.202091694, 0.112989739, 0.283432066, -0.0650387108, -0.154812038, -0.070825696, 0.0947837383, 0.0300658494, 0.147857964, -0.0216534138, 0.149756923, 0.0929859504, 0.0209971983, -0.00134888815, 0.0633148849, -0.0827424526, -0.000136449045, 0.19020921, -0.099270843, -0.0141247753, 0.0675853714, 0.0370295681, 0.183386773, -0.220024183, -0.0877708718, -0.214005783, -0.0824217796, -0.206398562, -0.221563339, -0.198710755, -0.119112119, -0.179287687, -0.00589003647, -0.145204052, 0.188346729, -0.233802795, 0.0376543291, -0.0215257984, -0.0865447745, 0.0118213641, 0.0664706305, -0.114263661, 0.0727500916, 0.0725146085, 0.189405486, 0.0885372013, -0.118517295, 0.0957777277, 0.113105021, -0.129922196, 0.0589649342, -0.0539315492, -0.0531233847, 0.0959037095, 0.159117237, 0.149913475, -0.0260760263, -0.0374908708, 0.105810463, 0.0345708914, 0.145390734, -0.0901318491, -0.0717779323, -0.0579015464, 0.0103023499, 0.205496356, 0.0216532797, -0.0160493869, 0.0679177195, -0.101879142, -0.0618111826, -0.0948672071, -0.0378079861, -0.0649976283, 0.0622105785, -0.0198299233, 0.117059089, 0.152212754, -0.112169929, 0.181148887, -0.168585852, 0.159860879, -0.0673378035, 0.0107045667, -0.0135089708, -0.0416479558, 0.0822456405, -0.127546847, -0.19231008, 0.173437029, 0.316009939, -0.185705617, -0.200298309, -0.158173889, 0.109854989, 0.152270272, 0.0278286487, 0.131128207, -0.071521163, 0.0525241606, 0.190306738, -0.124342375, 0.167207927, -0.0263414159, 0.0591874644, -0.0529713295, 0.0697124153, 0.054551594, -0.0173513144, -0.057966955, 0.0469674952, 0.178930059, -0.167295069, 0.0556705557, -0.217425913, 0.233187571, -0.0404247306, -0.173242241, 0.184321582, 0.102461167, -0.117671609, 0.0971307158, -0.212536231, -0.0653044954, -0.0705413967, 0.0569576286, 0.0243945643, 0.130107, -0.167852372, 0.0545675196, -0.238953099, 0.0423130803, 0.210260853, -0.0551566482, 0.26816833, 0.22665599, 0.225868911, -0.0444056578, -0.160370082, 0.0105681, -0.122951277, -0.115540609, -0.146256328, 0.188854426, 0.0384555124, -0.208536968, 0.277146548, 0.121490255, -0.0306008048, 0.0699297115, -0.22213009, 0.125744939, 0.205969438, 0.0161051843, -0.0934454426, 0.066526264, -0.123336747, 0.0589029752, 0.0126853334, 0.0986614898, -0.161116496, 0.0941702724, 0.0936794654, 0.196723357, 0.115641594, -0.157700956, 0.189485446, 0.114763916, -0.0271968227, 0.113643214, 0.195243552, 0.0987473726, 0.0990002304, -0.103220224, -0.150364637, 0.103585221, 0.107007116, 0.135821953, 0.181942925, -0.0627690554, -0.144740254, -0.109147213, -0.197329372, 0.0922926366, -0.163006827, 0.176730946, -0.122540452, -0.0845109373, 0.0133600179, 0.192756966, 0.1442388, 0.0578771867, -0.193552926, -0.110479511, -0.139845818, -0.165370867, -0.193599299, 0.20830974, 0.0628420413, 0.0663306862, 0.0201054998, -0.165055826, -0.00232632901, 0.0501528941, -0.162904873, 0.0240556058, -0.224557728, -0.207684785, -0.167241246, 0.0520122238, -0.150205687, -0.0774307996, 0.11285919, -0.0143467495, -0.0623829924, -0.0121905468, 0.149959132, -0.143484727, -0.241820574, 0.0834508464, 0.260972261, -0.0260955114, 0.24016428, -0.0213887114, 0.187113076, -0.0581168793, -0.0142169902, 0.12647666, -0.12786144, 0.167034611, 0.279815257, -0.179704726, 0.0132486979, 0.306648284, 0.178435475, -0.171064615, 0.0263747424, -0.0204333719, 0.21583344, 0.0672153682, -0.00418544794, 0.273084223, 0.157282963, -0.227137044, -0.136186168, -0.110910267, -0.12844494, 0.221502915, 0.213847071, 0.13926363, 0.259363115, -0.0436799936, 0.129494667, -0.0956437588, -0.247783363, 0.0357580781, 0.190545321, 0.139593437, 0.301190645, -0.155897871, 0.211046383, 0.180168241, -0.0615664087, 0.0724108592, -0.0146866199, -0.00990192872, 0.174645156, -0.0571350642, 0.0744009539, 0.148385659, -0.0929297581, -0.0392975882, 0.173364505, 0.0863989219, -0.111795798, 0.2648094, 0.0697908551, 0.0017024983, 0.000772171537, -0.191161424, -0.189653471, -0.0896795243, -0.0889835954, 0.120452896, 0.0736927539, 0.134213611, 0.205259874, -0.130877107, 0.180374101, -0.157959193, 0.176034316, 0.0191567838, 0.0846825391, -0.108345933, 0.202308819, -0.119057111, -0.198355615, -0.106700107, -0.0142671615, -0.0904524177, -0.136138856, 0.207652286, 0.154344276, 0.0967385918, 0.0491920561, 0.0370327979, 0.113051429, -0.198209167, -0.210644111, 0.100362405, -0.00893753767, 0.160789892, 0.0860281438, 0.149556741, -0.120294005, 0.0554995388, -0.189491674, -0.216242567, 0.164922521, -0.0101215243, 0.163655207, -0.209463686, 0.153605536, 0.135718778, -0.0541202426, 0.0377530009, -0.147346109, 0.138376907, 0.214301333, 0.10419561, 0.00336061418, 0.062403366, 0.142508909, 0.1622089, 0.136284068, 0.133917317, -0.179188401, 0.166013911, -0.162876546, 0.182987556, -0.101054475, 0.207223997, -0.100585461, 0.108998492, -0.059228152, -0.289831012, -0.0246569235, -0.00949376542, 0.175843939, -0.00427034125, 0.133596122, -0.0528981984, 0.174341112, -0.323382407, -0.0103142979, 0.0814552531, -0.0453974083, 0.0312591642, -0.0158383772, 0.018919412, -0.0416506566, -0.0423595347, 0.104281411, 0.125730589, 0.167497084, 0.190087736, 0.0710149929, 0.0990974009, -0.117281586, 0.103747696, 0.119485021, -0.0836957917, -0.219795361, -0.000133946538, -0.115642637, -0.0691571683, 0.00982022285, -0.128957704, 0.252099067, 0.190815985, 0.156464547, 0.0271001942, 0.12782681, -0.18666859, -0.100569583, -0.115921304, 0.245715797, 0.0163808819, 0.113201968, 0.270258486, 0.0548837595, 0.103501529, 0.170653298, 0.106830947, 0.0374602042, 0.227922827, -0.00101049035, 0.154585198, 0.0332156345, 0.00934819411, -0.0605532117, 0.00581356371, 0.247514546, 0.257806003, 0.10757257, 0.150476232, 0.0365517661, 0.0860407799, -0.145575255];
